	WAMANAGER_CICLO_PRELIEVO_PALL_RUN:
		IF Mission^.State = MISSION_STATE_NOP OR Mission^.State = MISSION_STATE_DEPOSITO_FALDA_END THEN
			QuotaFuoriIngombro_Z_AVUOTO_CCENTRALE := 0;
			QuotaFuoriIngombro_Z_ConPALLET := 0;
			(* Valuto gli ostacoli *)	
			FOR f:=1 TO MAXFOOTPRINT DO	
				IF QuotaFuoriIngombro_Z_AVUOTO_CCENTRALE <= WorkFootPrint^[f].Z + WorkFootPrint^[f].ZDim + TCPParameter.Z + OffsetSicurezza.Avuoto THEN
					QuotaFuoriIngombro_Z_AVUOTO_CCENTRALE := WorkFootPrint^[f].Z + WorkFootPrint^[f].ZDim + TCPParameter.Z + OffsetSicurezza.Avuoto;
				END_IF
				IF Mission^.TPick = TPICK_PALLET THEN
					IF QuotaFuoriIngombro_Z_ConPALLET <= WorkFootPrint^[f].Z + WorkFootPrint^[f].ZDim + Dimensione_Z_ElementoInPresaX_Ingombro + OffsetSicurezza.ConPallet THEN
						QuotaFuoriIngombro_Z_ConPALLET := WorkFootPrint^[f].Z + WorkFootPrint^[f].ZDim + Dimensione_Z_ElementoInPresaX_Ingombro + OffsetSicurezza.ConPallet;
					END_IF
				END_IF
			END_FOR
			(* Valuto le aree *)
			FOR a:=1 TO MAXAREA DO
				AltezzaDiIngombroArea_CCENTRALE := 0;
				IF WorkAreaState^[a].H > WorkAreaState^[a].HPL THEN
					AltezzaDiIngombroArea_CCENTRALE := WorkAreaState^[a].H;
				ELSE
					AltezzaDiIngombroArea_CCENTRALE := WorkAreaState^[a].HPL;
				END_IF
				(* Se ho la postazione falde e/o catasta vuoti con riscontri fissi metto la quota fissa di altezza della postazione all'altezza massima*)
				IF WorkArea^[a].Typology = TYPOLOGY_LAYER THEN
					AltezzaDiIngombroArea_CCENTRALE := ALTEZZA_CATASTA_FALDE;
				ELSIF  WorkArea^[a].Typology <> TYPOLOGY_STACK AND CATASTA_VUOTI_CON_RISCONTRI_FISSI THEN
					AltezzaDiIngombroArea_CCENTRALE := ALTEZZA_CATASTA_VUOTI;
				END_IF
				IF QuotaFuoriIngombro_Z_AVUOTO_CCENTRALE <= AltezzaDiIngombroArea_CCENTRALE + TCPParameter.Z + OffsetSicurezza.Avuoto THEN
					QuotaFuoriIngombro_Z_AVUOTO_CCENTRALE := AltezzaDiIngombroArea_CCENTRALE + TCPParameter.Z + OffsetSicurezza.Avuoto;
				END_IF
				IF QuotaFuoriIngombro_Z_ConPALLET <= AltezzaDiIngombroArea_CCENTRALE + Dimensione_Z_ElementoInPresaX_Ingombro + OffsetSicurezza.ConPallet THEN
					QuotaFuoriIngombro_Z_ConPALLET := AltezzaDiIngombroArea_CCENTRALE + Dimensione_Z_ElementoInPresaX_Ingombro + OffsetSicurezza.ConPallet;
				END_IF
			END_FOR
			(* Valuto I Pick-Point *)
			(*CASE TIPO_RIBALTINO OF
				RIBALTINO_DOPO_SQUADRO:
					FOR P:=1 TO MAXPICKPOINT DO
						AltezzaDiIngombroPuntiPrelievo := 0;
						IF  WorkPickPoint^[P].Zh + WorkPickPointState^[P].ZDim >= WorkPickPointDimension[P].Zdim THEN // Se Altezza orrizzontale Ribaltino + Zpacco >= Ingombro Verticale Ribaltino
							AltezzaDiIngombroPuntiPrelievo := WorkPickPoint^[P].Zh + WorkPickPointState^[P].ZDim;
						END_IF
						IF WorkPickPoint^[P].Zv + WorkPickPointState^[P].ZTilter + WorkPickPointState^[P].YDim >= WorkPickPointDimension[P].Zdim THEN // Se Altezza Vertivale Ribaltino + Quota Fermo + Ypacco >= Ingombro Verticale Ribaltino
							AltezzaDiIngombroPuntiPrelievo := WorkPickPoint^[P].Zv + WorkPickPointState^[P].ZTilter + WorkPickPointState^[P].YDim;
						END_IF
						IF WorkPickPointDimension[P].Zdim >= AltezzaDiIngombroPuntiPrelievo THEN //Se Ingombro Verticale Ribaltino >= Dell'ingombro valutato sopra
							AltezzaDiIngombroPuntiPrelievo := WorkPickPointDimension[P].Zdim;
						END_IF
						IF QuotaFuoriIngombro_Z_AVUOTO_CCENTRALE <= AltezzaDiIngombroPuntiPrelievo + TCPParameter.Z + OffsetSicurezza.Avuoto THEN //Se Quota fuori ingombro <= dell' ingombro del punto di prelievo
							QuotaFuoriIngombro_Z_AVUOTO_CCENTRALE := AltezzaDiIngombroPuntiPrelievo + TCPParameter.Z + OffsetSicurezza.Avuoto;
						END_IF				
					END_FOR
				RIBALTINO_DIRETTO :
					FOR P:=1 TO MAXPICKPOINT DO
						AltezzaDiIngombroPuntiPrelievo := 0;
						IF  WorkPickPoint^[P].Zh + WorkPickPointState^[P].ZDim >= WorkPickPointDimension[P].Zdim THEN // Se Altezza orrizzontale Ribaltino + Zpacco >= Ingombro Verticale Ribaltino
							AltezzaDiIngombroPuntiPrelievo := WorkPickPoint^[P].Zh + WorkPickPointState^[P].ZDim;
						END_IF
						IF WorkPickPoint^[P].Zv + WorkPickPointState^[P].ZTilter + WorkPickPointState^[P].XDim >= WorkPickPointDimension[P].Zdim THEN // Se Altezza Vertivale Ribaltino + Quota Fermo + Ypacco >= Ingombro Verticale Ribaltino
							AltezzaDiIngombroPuntiPrelievo := WorkPickPoint^[P].Zv + WorkPickPointState^[P].ZTilter + WorkPickPointState^[P].XDim;
						END_IF
						IF WorkPickPointDimension[P].Zdim >= AltezzaDiIngombroPuntiPrelievo THEN //Se Ingombro Verticale Ribaltino >= Dell'ingombro valutato sopra
							AltezzaDiIngombroPuntiPrelievo := WorkPickPointDimension[P].Zdim;
						END_IF
						IF QuotaFuoriIngombro_Z_AVUOTO_CCENTRALE <= AltezzaDiIngombroPuntiPrelievo + TCPParameter.Z + OffsetSicurezza.Avuoto THEN //Se Quota fuori ingombro <= dell' ingombro del punto di prelievo
							QuotaFuoriIngombro_Z_AVUOTO_CCENTRALE := AltezzaDiIngombroPuntiPrelievo + TCPParameter.Z + OffsetSicurezza.Avuoto;
						END_IF				
					END_FOR
			END_CASE*)
			
			(*IF Mission^.TPick = TPICK_PALLET THEN
				Traiettoria^.PassModePoint_Z_Enable[1] := TRUE; // traslazione verso l'alto e verticale.....inizio degli altri movimenti 200 mm prima dela fine
				Traiettoria^.PassModePoint_Z[1] := QuotaFuoriIngombro_Z_AVUOTO_CCENTRALE - OffsetPassMode.Z;
				Traiettoria^.PassModePoint_X_Enable[1] := TRUE;	
				IF ModuleAX_X^.Ax^.Status.ActPosition >= Mission^.XPick THEN			// se la posizione attuale in X è MAGGIORE della posizione di destinazione
					Traiettoria^.PassModePoint_X[1] := Mission^.XPick + OffsetPassMode.X;			
				ELSE																	// se la posizione attuale in X è MINORE della posizione di destinazione
					Traiettoria^.PassModePoint_X[1] := Mission^.XPick - OffsetPassMode.X;			
				END_IF			
				Traiettoria^.PassModePoint_Y_Enable[1] := TRUE;
				Traiettoria^.PassModePoint_Y[1] := 0;			// inizio degli altri movimenti in corrispondenza della posizione attuale
				Traiettoria^.PassModePoint_J_Enable[1] := TRUE;
				Traiettoria^.PassModePoint_J[1] := 0;			// inizio degli altri movimenti in corrispondenza della posizione attuale
				Traiettoria^.PassModePoint_K_Enable[1] := TRUE;
				Traiettoria^.PassModePoint_K[1] := 0;			// inizio degli altri movimenti in corrispondenza della posizione attuale
			END_IF*)
		END_IF //riferito all'IF dello stato della missione	
														
	WAMANAGER_CICLO_PRELIEVO_PALL_END,						
		
	WAMANAGER_CICLO_DEPOSITO_PALL_RUN:
		IF Mission^.State = MISSION_STATE_NOP OR Mission^.State = MISSION_STATE_PRELIEVO_PALLET_END THEN
			QuotaFuoriIngombro_Z_AVUOTO_CCENTRALE := 0;
			QuotaFuoriIngombro_Z_ConPALLET := 0;
			(* Valuto gli ostacoli x la quota fuori ingombro*)	
			FOR f:=1 TO MAXFOOTPRINT DO	
				IF QuotaFuoriIngombro_Z_AVUOTO_CCENTRALE <= WorkFootPrint^[f].Z + WorkFootPrint^[f].ZDim + TCPParameter.Z + OffsetSicurezza.Avuoto THEN
					QuotaFuoriIngombro_Z_AVUOTO_CCENTRALE := WorkFootPrint^[f].Z + WorkFootPrint^[f].ZDim + TCPParameter.Z + OffsetSicurezza.Avuoto;
				END_IF
				IF QuotaFuoriIngombro_Z_ConPALLET <= WorkFootPrint^[f].Z + WorkFootPrint^[f].ZDim + Dimensione_Z_ElementoInPresaX_Ingombro + OffsetSicurezza.ConPallet THEN
					QuotaFuoriIngombro_Z_ConPALLET := WorkFootPrint^[f].Z + WorkFootPrint^[f].ZDim + Dimensione_Z_ElementoInPresaX_Ingombro + OffsetSicurezza.ConPallet;
				END_IF
			END_FOR
			(* Valuto le aree x la quota fuori ingombro *)
			FOR a:=1 TO MAXAREA DO
				AltezzaDiIngombroArea_CCENTRALE := 0;
				IF WorkAreaState^[a].H > WorkAreaState^[a].HPL THEN
					AltezzaDiIngombroArea_CCENTRALE := WorkAreaState^[a].H;
				ELSE
					AltezzaDiIngombroArea_CCENTRALE := WorkAreaState^[a].HPL;
				END_IF
				(* Se ho la postazione falde e/o catasta vuoti con riscontri fissi metto la quota fissa di altezza della postazione all'altezza massima*)
				IF WorkArea^[a].Typology = TYPOLOGY_LAYER THEN
					AltezzaDiIngombroArea_CCENTRALE := ALTEZZA_CATASTA_FALDE;
				ELSIF  WorkArea^[a].Typology <> TYPOLOGY_STACK AND CATASTA_VUOTI_CON_RISCONTRI_FISSI THEN
					AltezzaDiIngombroArea_CCENTRALE := ALTEZZA_CATASTA_VUOTI;
				END_IF
				IF QuotaFuoriIngombro_Z_AVUOTO_CCENTRALE <= AltezzaDiIngombroArea_CCENTRALE + TCPParameter.Z + OffsetSicurezza.Avuoto THEN
					QuotaFuoriIngombro_Z_AVUOTO_CCENTRALE := AltezzaDiIngombroArea_CCENTRALE + TCPParameter.Z + OffsetSicurezza.Avuoto;
				END_IF
				IF QuotaFuoriIngombro_Z_ConPALLET <= AltezzaDiIngombroArea_CCENTRALE + Dimensione_Z_ElementoInPresaX_Ingombro + OffsetSicurezza.ConPallet THEN
					QuotaFuoriIngombro_Z_ConPALLET := AltezzaDiIngombroArea_CCENTRALE + Dimensione_Z_ElementoInPresaX_Ingombro + OffsetSicurezza.ConPallet;
				END_IF
			END_FOR
			(* Valuto I Pick-Point *)
			(* Valuto I Pick-Point *)
			(*CASE TIPO_RIBALTINO OF
				RIBALTINO_DOPO_SQUADRO:
					FOR P:=1 TO MAXPICKPOINT DO
						AltezzaDiIngombroPuntiPrelievo := 0;
						IF  WorkPickPoint^[P].Zh + WorkPickPointState^[P].ZDim >= WorkPickPointDimension[P].Zdim THEN // Se Altezza orrizzontale Ribaltino + Zpacco >= Ingombro Verticale Ribaltino
							AltezzaDiIngombroPuntiPrelievo := WorkPickPoint^[P].Zh + WorkPickPointState^[P].ZDim;
						END_IF
						IF WorkPickPoint^[P].Zv + WorkPickPointState^[P].ZTilter + WorkPickPointState^[P].YDim >= WorkPickPointDimension[P].Zdim THEN // Se Altezza Vertivale Ribaltino + Quota Fermo + Ypacco >= Ingombro Verticale Ribaltino
							AltezzaDiIngombroPuntiPrelievo := WorkPickPoint^[P].Zv + WorkPickPointState^[P].ZTilter + WorkPickPointState^[P].YDim;
						END_IF
						IF WorkPickPointDimension[P].Zdim >= AltezzaDiIngombroPuntiPrelievo THEN //Se Ingombro Verticale Ribaltino >= Dell'ingombro valutato sopra
							AltezzaDiIngombroPuntiPrelievo := WorkPickPointDimension[P].Zdim;
						END_IF
						IF QuotaFuoriIngombro_Z_AVUOTO_CCENTRALE <= AltezzaDiIngombroPuntiPrelievo + TCPParameter.Z + OffsetSicurezza.Avuoto THEN //Se Quota fuori ingombro <= dell' ingombro del punto di prelievo
							QuotaFuoriIngombro_Z_AVUOTO_CCENTRALE := AltezzaDiIngombroPuntiPrelievo + TCPParameter.Z + OffsetSicurezza.Avuoto;
						END_IF
						IF QuotaFuoriIngombro_Z_ConPALLET <= AltezzaDiIngombroPuntiPrelievo + TCPParameter.Z + OffsetSicurezza.ConPallet THEN //Se Quota fuori ingombro <= dell' ingombro del punto di prelievo
							QuotaFuoriIngombro_Z_ConPALLET := AltezzaDiIngombroPuntiPrelievo + TCPParameter.Z + OffsetSicurezza.ConPallet;
						END_IF
					END_FOR
				RIBALTINO_DIRETTO :
					FOR P:=1 TO MAXPICKPOINT DO
						AltezzaDiIngombroPuntiPrelievo := 0;
						IF  WorkPickPoint^[P].Zh + WorkPickPointState^[P].ZDim >= WorkPickPointDimension[P].Zdim THEN // Se Altezza orrizzontale Ribaltino + Zpacco >= Ingombro Verticale Ribaltino
							AltezzaDiIngombroPuntiPrelievo := WorkPickPoint^[P].Zh + WorkPickPointState^[P].ZDim;
						END_IF
						IF WorkPickPoint^[P].Zv + WorkPickPointState^[P].ZTilter + WorkPickPointState^[P].XDim >= WorkPickPointDimension[P].Zdim THEN // Se Altezza Vertivale Ribaltino + Quota Fermo + Ypacco >= Ingombro Verticale Ribaltino
							AltezzaDiIngombroPuntiPrelievo := WorkPickPoint^[P].Zv + WorkPickPointState^[P].ZTilter + WorkPickPointState^[P].XDim;
						END_IF
						IF WorkPickPointDimension[P].Zdim >= AltezzaDiIngombroPuntiPrelievo THEN //Se Ingombro Verticale Ribaltino >= Dell'ingombro valutato sopra
							AltezzaDiIngombroPuntiPrelievo := WorkPickPointDimension[P].Zdim;
						END_IF
						IF QuotaFuoriIngombro_Z_AVUOTO_CCENTRALE <= AltezzaDiIngombroPuntiPrelievo + TCPParameter.Z + OffsetSicurezza.Avuoto THEN //Se Quota fuori ingombro <= dell' ingombro del punto di prelievo
							QuotaFuoriIngombro_Z_AVUOTO_CCENTRALE := AltezzaDiIngombroPuntiPrelievo + TCPParameter.Z + OffsetSicurezza.Avuoto;
						END_IF	
						IF QuotaFuoriIngombro_Z_ConPALLET <= AltezzaDiIngombroPuntiPrelievo + TCPParameter.Z + OffsetSicurezza.ConPallet THEN //Se Quota fuori ingombro <= dell' ingombro del punto di prelievo
							QuotaFuoriIngombro_Z_ConPALLET := AltezzaDiIngombroPuntiPrelievo + TCPParameter.Z + OffsetSicurezza.ConPallet;
						END_IF			
					END_FOR
			END_CASE*)
					
		END_IF //riferito all'IF dello stato della missione	
		
			
	WAMANAGER_CICLO_DEPOSITO_PALL_END,
	
	WAMANAGER_CICLO_FALDA_VUOTI_INIT,
	
	WAMANAGER_CICLO_PRELIEVO_FALDA_VUOTI_RUN:
		IF Mission^.State = MISSION_STATE_NOP THEN
			QuotaFuoriIngombro_Z_AVUOTO_CCENTRALE := 0;
			QuotaFuoriIngombro_Z_ConFALDA := 0;
			(* Valuto gli ostacoli *)	
			FOR f:=1 TO MAXFOOTPRINT DO	
				IF QuotaFuoriIngombro_Z_AVUOTO_CCENTRALE <= WorkFootPrint^[f].Z + WorkFootPrint^[f].ZDim + TCPParameter.Z + OffsetSicurezza.Avuoto THEN
					QuotaFuoriIngombro_Z_AVUOTO_CCENTRALE := WorkFootPrint^[f].Z + WorkFootPrint^[f].ZDim + TCPParameter.Z + OffsetSicurezza.Avuoto;
				END_IF
			END_FOR
			(* Valuto le aree *)
			FOR a:=1 TO MAXAREA DO
				AltezzaDiIngombroArea_CCENTRALE := 0;
				IF WorkAreaState^[a].H > WorkAreaState^[a].HPL THEN
					AltezzaDiIngombroArea_CCENTRALE := WorkAreaState^[a].H;
				ELSE
					AltezzaDiIngombroArea_CCENTRALE := WorkAreaState^[a].HPL;
				END_IF
				(* Se ho la postazione falde e/o catasta vuoti con riscontri fissi metto la quota fissa di altezza della postazione all'altezza massima*)
				IF WorkArea^[a].Typology = TYPOLOGY_LAYER THEN
					AltezzaDiIngombroArea_CCENTRALE := ALTEZZA_CATASTA_FALDE;
				ELSIF  WorkArea^[a].Typology <> TYPOLOGY_STACK AND CATASTA_VUOTI_CON_RISCONTRI_FISSI THEN
					AltezzaDiIngombroArea_CCENTRALE := ALTEZZA_CATASTA_VUOTI;
				END_IF
				IF QuotaFuoriIngombro_Z_AVUOTO_CCENTRALE <= AltezzaDiIngombroArea_CCENTRALE + TCPParameter.Z + OffsetSicurezza.Avuoto THEN
					QuotaFuoriIngombro_Z_AVUOTO_CCENTRALE := AltezzaDiIngombroArea_CCENTRALE + TCPParameter.Z + OffsetSicurezza.Avuoto;
				END_IF
			END_FOR
			(* Valuto I Pick-Point *)
			(*CASE TIPO_RIBALTINO OF
				RIBALTINO_DOPO_SQUADRO:
					FOR P:=1 TO MAXPICKPOINT DO
						AltezzaDiIngombroPuntiPrelievo := 0;
						IF  WorkPickPoint^[P].Zh + WorkPickPointState^[P].ZDim >= WorkPickPointDimension[P].Zdim THEN // Se Altezza orrizzontale Ribaltino + Zpacco >= Ingombro Verticale Ribaltino
							AltezzaDiIngombroPuntiPrelievo := WorkPickPoint^[P].Zh + WorkPickPointState^[P].ZDim;
						END_IF
						IF WorkPickPoint^[P].Zv + WorkPickPointState^[P].ZTilter + WorkPickPointState^[P].YDim >= WorkPickPointDimension[P].Zdim THEN // Se Altezza Vertivale Ribaltino + Quota Fermo + Ypacco >= Ingombro Verticale Ribaltino
							AltezzaDiIngombroPuntiPrelievo := WorkPickPoint^[P].Zv + WorkPickPointState^[P].ZTilter + WorkPickPointState^[P].YDim;
						END_IF
						IF WorkPickPointDimension[P].Zdim >= AltezzaDiIngombroPuntiPrelievo THEN //Se Ingombro Verticale Ribaltino >= Dell'ingombro valutato sopra
							AltezzaDiIngombroPuntiPrelievo := WorkPickPointDimension[P].Zdim;
						END_IF
						IF QuotaFuoriIngombro_Z_AVUOTO_CCENTRALE <= AltezzaDiIngombroPuntiPrelievo + TCPParameter.Z + OffsetSicurezza.Avuoto THEN //Se Quota fuori ingombro <= dell' ingombro del punto di prelievo
							QuotaFuoriIngombro_Z_AVUOTO_CCENTRALE := AltezzaDiIngombroPuntiPrelievo + TCPParameter.Z + OffsetSicurezza.Avuoto;
						END_IF				
					END_FOR
				RIBALTINO_DIRETTO :
					FOR P:=1 TO MAXPICKPOINT DO
						AltezzaDiIngombroPuntiPrelievo := 0;
						IF  WorkPickPoint^[P].Zh + WorkPickPointState^[P].ZDim >= WorkPickPointDimension[P].Zdim THEN // Se Altezza orrizzontale Ribaltino + Zpacco >= Ingombro Verticale Ribaltino
							AltezzaDiIngombroPuntiPrelievo := WorkPickPoint^[P].Zh + WorkPickPointState^[P].ZDim;
						END_IF
						IF WorkPickPoint^[P].Zv + WorkPickPointState^[P].ZTilter + WorkPickPointState^[P].XDim >= WorkPickPointDimension[P].Zdim THEN // Se Altezza Vertivale Ribaltino + Quota Fermo + Ypacco >= Ingombro Verticale Ribaltino
							AltezzaDiIngombroPuntiPrelievo := WorkPickPoint^[P].Zv + WorkPickPointState^[P].ZTilter + WorkPickPointState^[P].XDim;
						END_IF
						IF WorkPickPointDimension[P].Zdim >= AltezzaDiIngombroPuntiPrelievo THEN //Se Ingombro Verticale Ribaltino >= Dell'ingombro valutato sopra
							AltezzaDiIngombroPuntiPrelievo := WorkPickPointDimension[P].Zdim;
						END_IF
						IF QuotaFuoriIngombro_Z_AVUOTO_CCENTRALE <= AltezzaDiIngombroPuntiPrelievo + TCPParameter.Z + OffsetSicurezza.Avuoto THEN //Se Quota fuori ingombro <= dell' ingombro del punto di prelievo
							QuotaFuoriIngombro_Z_AVUOTO_CCENTRALE := AltezzaDiIngombroPuntiPrelievo + TCPParameter.Z + OffsetSicurezza.Avuoto;
						END_IF				
					END_FOR
			END_CASE*)
			QuotaFuoriIngombro_Z_ConFALDA := QuotaFuoriIngombro_Z_AVUOTO_CCENTRALE;
			
		END_IF //riferito all'IF dello stato della missione	
					
	WAMANAGER_CICLO_PRELIEVO_FALDA_VUOTI_END,
		
	WAMANAGER_CICLO_DEPOSITO_FALDA_VUOTI_RUN:
		IF Mission^.State = MISSION_STATE_NOP OR Mission^.State = MISSION_STATE_PRELIEVO_FALDA_END THEN
			QuotaFuoriIngombro_Z_AVUOTO_CCENTRALE := 0;
			QuotaFuoriIngombro_Z_ConFALDA := 0;
			(* Valuto gli ostacoli *)	
			FOR f:=1 TO MAXFOOTPRINT DO	
				IF QuotaFuoriIngombro_Z_AVUOTO_CCENTRALE <= WorkFootPrint^[f].Z + WorkFootPrint^[f].ZDim + TCPParameter.Z + OffsetSicurezza.Avuoto THEN
					QuotaFuoriIngombro_Z_AVUOTO_CCENTRALE := WorkFootPrint^[f].Z + WorkFootPrint^[f].ZDim + TCPParameter.Z + OffsetSicurezza.Avuoto;
				END_IF
			END_FOR
			(* Valuto le aree *)
			FOR a:=1 TO MAXAREA DO
				AltezzaDiIngombroArea_CCENTRALE := 0;
				IF WorkAreaState^[a].H > WorkAreaState^[a].HPL THEN
					AltezzaDiIngombroArea_CCENTRALE := WorkAreaState^[a].H;
				ELSE
					AltezzaDiIngombroArea_CCENTRALE := WorkAreaState^[a].HPL;
				END_IF
				(* Se ho la postazione falde e/o catasta vuoti con riscontri fissi metto la quota fissa di altezza della postazione all'altezza massima*)
				IF WorkArea^[a].Typology = TYPOLOGY_LAYER THEN
					AltezzaDiIngombroArea_CCENTRALE := ALTEZZA_CATASTA_FALDE;
				ELSIF  WorkArea^[a].Typology <> TYPOLOGY_STACK AND CATASTA_VUOTI_CON_RISCONTRI_FISSI THEN
					AltezzaDiIngombroArea_CCENTRALE := ALTEZZA_CATASTA_VUOTI;
				END_IF
				IF QuotaFuoriIngombro_Z_AVUOTO_CCENTRALE <= AltezzaDiIngombroArea_CCENTRALE + TCPParameter.Z + OffsetSicurezza.Avuoto THEN
					QuotaFuoriIngombro_Z_AVUOTO_CCENTRALE := AltezzaDiIngombroArea_CCENTRALE + TCPParameter.Z + OffsetSicurezza.Avuoto;
				END_IF
			END_FOR
			(* Valuto I Pick-Point *)
			(*CASE TIPO_RIBALTINO OF
				RIBALTINO_DOPO_SQUADRO:
					FOR P:=1 TO MAXPICKPOINT DO
						AltezzaDiIngombroPuntiPrelievo := 0;
						IF  WorkPickPoint^[P].Zh + WorkPickPointState^[P].ZDim >= WorkPickPointDimension[P].Zdim THEN // Se Altezza orrizzontale Ribaltino + Zpacco >= Ingombro Verticale Ribaltino
							AltezzaDiIngombroPuntiPrelievo := WorkPickPoint^[P].Zh + WorkPickPointState^[P].ZDim;
						END_IF
						IF WorkPickPoint^[P].Zv + WorkPickPointState^[P].ZTilter + WorkPickPointState^[P].YDim >= WorkPickPointDimension[P].Zdim THEN // Se Altezza Vertivale Ribaltino + Quota Fermo + Ypacco >= Ingombro Verticale Ribaltino
							AltezzaDiIngombroPuntiPrelievo := WorkPickPoint^[P].Zv + WorkPickPointState^[P].ZTilter + WorkPickPointState^[P].YDim;
						END_IF
						IF WorkPickPointDimension[P].Zdim >= AltezzaDiIngombroPuntiPrelievo THEN //Se Ingombro Verticale Ribaltino >= Dell'ingombro valutato sopra
							AltezzaDiIngombroPuntiPrelievo := WorkPickPointDimension[P].Zdim;
						END_IF
						IF QuotaFuoriIngombro_Z_AVUOTO_CCENTRALE <= AltezzaDiIngombroPuntiPrelievo + TCPParameter.Z + OffsetSicurezza.Avuoto THEN //Se Quota fuori ingombro <= dell' ingombro del punto di prelievo
							QuotaFuoriIngombro_Z_AVUOTO_CCENTRALE := AltezzaDiIngombroPuntiPrelievo + TCPParameter.Z + OffsetSicurezza.Avuoto;
						END_IF				
					END_FOR
				RIBALTINO_DIRETTO :
					FOR P:=1 TO MAXPICKPOINT DO
						AltezzaDiIngombroPuntiPrelievo := 0;
						IF  WorkPickPoint^[P].Zh + WorkPickPointState^[P].ZDim >= WorkPickPointDimension[P].Zdim THEN // Se Altezza orrizzontale Ribaltino + Zpacco >= Ingombro Verticale Ribaltino
							AltezzaDiIngombroPuntiPrelievo := WorkPickPoint^[P].Zh + WorkPickPointState^[P].ZDim;
						END_IF
						IF WorkPickPoint^[P].Zv + WorkPickPointState^[P].ZTilter + WorkPickPointState^[P].XDim >= WorkPickPointDimension[P].Zdim THEN // Se Altezza Vertivale Ribaltino + Quota Fermo + Ypacco >= Ingombro Verticale Ribaltino
							AltezzaDiIngombroPuntiPrelievo := WorkPickPoint^[P].Zv + WorkPickPointState^[P].ZTilter + WorkPickPointState^[P].XDim;
						END_IF
						IF WorkPickPointDimension[P].Zdim >= AltezzaDiIngombroPuntiPrelievo THEN //Se Ingombro Verticale Ribaltino >= Dell'ingombro valutato sopra
							AltezzaDiIngombroPuntiPrelievo := WorkPickPointDimension[P].Zdim;
						END_IF
						IF QuotaFuoriIngombro_Z_AVUOTO_CCENTRALE <= AltezzaDiIngombroPuntiPrelievo + TCPParameter.Z + OffsetSicurezza.Avuoto THEN //Se Quota fuori ingombro <= dell' ingombro del punto di prelievo
							QuotaFuoriIngombro_Z_AVUOTO_CCENTRALE := AltezzaDiIngombroPuntiPrelievo + TCPParameter.Z + OffsetSicurezza.Avuoto;
						END_IF				
					END_FOR
			END_CASE*)
			QuotaFuoriIngombro_Z_ConFALDA := QuotaFuoriIngombro_Z_AVUOTO_CCENTRALE;
			
		END_IF //riferito all'IF dello stato della missione	
									
	WAMANAGER_CICLO_DEPOSITO_FALDA_VUOTI_END,*)
	
	WAMANAGER_CICLO_FALDA_INIT,
	
	WAMANAGER_CICLO_PRELIEVO_FALDA_RUN:
		IF Mission^.State = MISSION_STATE_NOP THEN
			QuotaFuoriIngombro_Z_AVUOTO_CCENTRALE := 0;
			QuotaFuoriIngombro_Z_ConFALDA := 0;
			(* Valuto gli ostacoli *)	
			FOR f:=1 TO MAXFOOTPRINT DO	
				IF QuotaFuoriIngombro_Z_AVUOTO_CCENTRALE <= WorkFootPrint^[f].Z + WorkFootPrint^[f].ZDim + TCPParameter.Z + OffsetSicurezza.Avuoto THEN
					QuotaFuoriIngombro_Z_AVUOTO_CCENTRALE := WorkFootPrint^[f].Z + WorkFootPrint^[f].ZDim + TCPParameter.Z + OffsetSicurezza.Avuoto;
				END_IF
			END_FOR
			(* Valuto le aree *)
			FOR a:=1 TO MAXAREA DO
				AltezzaDiIngombroArea_CCENTRALE := 0;
				IF WorkAreaState^[a].H > WorkAreaState^[a].HPL THEN
					AltezzaDiIngombroArea_CCENTRALE := WorkAreaState^[a].H;
				ELSE
					AltezzaDiIngombroArea_CCENTRALE := WorkAreaState^[a].HPL;
				END_IF
				IF QuotaFuoriIngombro_Z_AVUOTO_CCENTRALE <= AltezzaDiIngombroArea_CCENTRALE + TCPParameter.Z + OffsetSicurezza.Avuoto THEN
					QuotaFuoriIngombro_Z_AVUOTO_CCENTRALE := AltezzaDiIngombroArea_CCENTRALE + TCPParameter.Z + OffsetSicurezza.Avuoto;
				END_IF
			END_FOR
			(* Valuto I Pick-Point *)
			(*CASE TIPO_RIBALTINO OF
				RIBALTINO_DOPO_SQUADRO:
					FOR P:=1 TO MAXPICKPOINT DO
						AltezzaDiIngombroPuntiPrelievo := 0;
						IF  WorkPickPoint^[P].Zh + WorkPickPointState^[P].ZDim >= WorkPickPointDimension[P].Zdim THEN // Se Altezza orrizzontale Ribaltino + Zpacco >= Ingombro Verticale Ribaltino
							AltezzaDiIngombroPuntiPrelievo := WorkPickPoint^[P].Zh + WorkPickPointState^[P].ZDim;
						END_IF
						IF WorkPickPoint^[P].Zv + WorkPickPointState^[P].ZTilter + WorkPickPointState^[P].YDim >= WorkPickPointDimension[P].Zdim THEN // Se Altezza Vertivale Ribaltino + Quota Fermo + Ypacco >= Ingombro Verticale Ribaltino
							AltezzaDiIngombroPuntiPrelievo := WorkPickPoint^[P].Zv + WorkPickPointState^[P].ZTilter + WorkPickPointState^[P].YDim;
						END_IF
						IF WorkPickPointDimension[P].Zdim >= AltezzaDiIngombroPuntiPrelievo THEN //Se Ingombro Verticale Ribaltino >= Dell'ingombro valutato sopra
							AltezzaDiIngombroPuntiPrelievo := WorkPickPointDimension[P].Zdim;
						END_IF
						IF QuotaFuoriIngombro_Z_AVUOTO_CCENTRALE <= AltezzaDiIngombroPuntiPrelievo + TCPParameter.Z + OffsetSicurezza.Avuoto THEN //Se Quota fuori ingombro <= dell' ingombro del punto di prelievo
							QuotaFuoriIngombro_Z_AVUOTO_CCENTRALE := AltezzaDiIngombroPuntiPrelievo + TCPParameter.Z + OffsetSicurezza.Avuoto;
						END_IF				
					END_FOR
				RIBALTINO_DIRETTO :
					FOR P:=1 TO MAXPICKPOINT DO
						AltezzaDiIngombroPuntiPrelievo := 0;
						IF  WorkPickPoint^[P].Zh + WorkPickPointState^[P].ZDim >= WorkPickPointDimension[P].Zdim THEN // Se Altezza orrizzontale Ribaltino + Zpacco >= Ingombro Verticale Ribaltino
							AltezzaDiIngombroPuntiPrelievo := WorkPickPoint^[P].Zh + WorkPickPointState^[P].ZDim;
						END_IF
						IF WorkPickPoint^[P].Zv + WorkPickPointState^[P].ZTilter + WorkPickPointState^[P].XDim >= WorkPickPointDimension[P].Zdim THEN // Se Altezza Vertivale Ribaltino + Quota Fermo + Ypacco >= Ingombro Verticale Ribaltino
							AltezzaDiIngombroPuntiPrelievo := WorkPickPoint^[P].Zv + WorkPickPointState^[P].ZTilter + WorkPickPointState^[P].XDim;
						END_IF
						IF WorkPickPointDimension[P].Zdim >= AltezzaDiIngombroPuntiPrelievo THEN //Se Ingombro Verticale Ribaltino >= Dell'ingombro valutato sopra
							AltezzaDiIngombroPuntiPrelievo := WorkPickPointDimension[P].Zdim;
						END_IF
						IF QuotaFuoriIngombro_Z_AVUOTO_CCENTRALE <= AltezzaDiIngombroPuntiPrelievo + TCPParameter.Z + OffsetSicurezza.Avuoto THEN //Se Quota fuori ingombro <= dell' ingombro del punto di prelievo
							QuotaFuoriIngombro_Z_AVUOTO_CCENTRALE := AltezzaDiIngombroPuntiPrelievo + TCPParameter.Z + OffsetSicurezza.Avuoto;
						END_IF				
					END_FOR
			END_CASE*)
			QuotaFuoriIngombro_Z_ConFALDA := QuotaFuoriIngombro_Z_AVUOTO_CCENTRALE;
			
		END_IF //riferito all'IF dello stato della missione	
																
	WAMANAGER_CICLO_PRELIEVO_FALDA_END,
			
	WAMANAGER_CICLO_DEPOSITO_FALDA_RUN:
		IF Mission^.State = MISSION_STATE_NOP OR Mission^.State = MISSION_STATE_PRELIEVO_FALDA_END THEN
			QuotaFuoriIngombro_Z_AVUOTO_CCENTRALE := 0;
			QuotaFuoriIngombro_Z_ConFALDA := 0;
			(* Valuto gli ostacoli *)	
			FOR f:=1 TO MAXFOOTPRINT DO	
				IF QuotaFuoriIngombro_Z_AVUOTO_CCENTRALE <= WorkFootPrint^[f].Z + WorkFootPrint^[f].ZDim + TCPParameter.Z + OffsetSicurezza.Avuoto THEN
					QuotaFuoriIngombro_Z_AVUOTO_CCENTRALE := WorkFootPrint^[f].Z + WorkFootPrint^[f].ZDim + TCPParameter.Z + OffsetSicurezza.Avuoto;
				END_IF
			END_FOR
			(* Valuto le aree *)
			FOR a:=1 TO MAXAREA DO
				AltezzaDiIngombroArea_CCENTRALE := 0;
				IF WorkAreaState^[a].H > WorkAreaState^[a].HPL THEN
					AltezzaDiIngombroArea_CCENTRALE := WorkAreaState^[a].H;
				ELSE
					AltezzaDiIngombroArea_CCENTRALE := WorkAreaState^[a].HPL;
				END_IF
				IF QuotaFuoriIngombro_Z_AVUOTO_CCENTRALE <= AltezzaDiIngombroArea_CCENTRALE + TCPParameter.Z + OffsetSicurezza.Avuoto THEN
					QuotaFuoriIngombro_Z_AVUOTO_CCENTRALE := AltezzaDiIngombroArea_CCENTRALE + TCPParameter.Z + OffsetSicurezza.Avuoto;
				END_IF
			END_FOR
			(* Valuto I Pick-Point *)
			(*CASE TIPO_RIBALTINO OF
				RIBALTINO_DOPO_SQUADRO:
					FOR P:=1 TO MAXPICKPOINT DO
						AltezzaDiIngombroPuntiPrelievo := 0;
						IF  WorkPickPoint^[P].Zh + WorkPickPointState^[P].ZDim >= WorkPickPointDimension[P].Zdim THEN // Se Altezza orrizzontale Ribaltino + Zpacco >= Ingombro Verticale Ribaltino
							AltezzaDiIngombroPuntiPrelievo := WorkPickPoint^[P].Zh + WorkPickPointState^[P].ZDim;
						END_IF
						IF WorkPickPoint^[P].Zv + WorkPickPointState^[P].ZTilter + WorkPickPointState^[P].YDim >= WorkPickPointDimension[P].Zdim THEN // Se Altezza Vertivale Ribaltino + Quota Fermo + Ypacco >= Ingombro Verticale Ribaltino
							AltezzaDiIngombroPuntiPrelievo := WorkPickPoint^[P].Zv + WorkPickPointState^[P].ZTilter + WorkPickPointState^[P].YDim;
						END_IF
						IF WorkPickPointDimension[P].Zdim >= AltezzaDiIngombroPuntiPrelievo THEN //Se Ingombro Verticale Ribaltino >= Dell'ingombro valutato sopra
							AltezzaDiIngombroPuntiPrelievo := WorkPickPointDimension[P].Zdim;
						END_IF
						IF QuotaFuoriIngombro_Z_AVUOTO_CCENTRALE <= AltezzaDiIngombroPuntiPrelievo + TCPParameter.Z + OffsetSicurezza.Avuoto THEN //Se Quota fuori ingombro <= dell' ingombro del punto di prelievo
							QuotaFuoriIngombro_Z_AVUOTO_CCENTRALE := AltezzaDiIngombroPuntiPrelievo + TCPParameter.Z + OffsetSicurezza.Avuoto;
						END_IF				
					END_FOR
				RIBALTINO_DIRETTO :
					FOR P:=1 TO MAXPICKPOINT DO
						AltezzaDiIngombroPuntiPrelievo := 0;
						IF  WorkPickPoint^[P].Zh + WorkPickPointState^[P].ZDim >= WorkPickPointDimension[P].Zdim THEN // Se Altezza orrizzontale Ribaltino + Zpacco >= Ingombro Verticale Ribaltino
							AltezzaDiIngombroPuntiPrelievo := WorkPickPoint^[P].Zh + WorkPickPointState^[P].ZDim;
						END_IF
						IF WorkPickPoint^[P].Zv + WorkPickPointState^[P].ZTilter + WorkPickPointState^[P].XDim >= WorkPickPointDimension[P].Zdim THEN // Se Altezza Vertivale Ribaltino + Quota Fermo + Ypacco >= Ingombro Verticale Ribaltino
							AltezzaDiIngombroPuntiPrelievo := WorkPickPoint^[P].Zv + WorkPickPointState^[P].ZTilter + WorkPickPointState^[P].XDim;
						END_IF
						IF WorkPickPointDimension[P].Zdim >= AltezzaDiIngombroPuntiPrelievo THEN //Se Ingombro Verticale Ribaltino >= Dell'ingombro valutato sopra
							AltezzaDiIngombroPuntiPrelievo := WorkPickPointDimension[P].Zdim;
						END_IF
						IF QuotaFuoriIngombro_Z_AVUOTO_CCENTRALE <= AltezzaDiIngombroPuntiPrelievo + TCPParameter.Z + OffsetSicurezza.Avuoto THEN //Se Quota fuori ingombro <= dell' ingombro del punto di prelievo
							QuotaFuoriIngombro_Z_AVUOTO_CCENTRALE := AltezzaDiIngombroPuntiPrelievo + TCPParameter.Z + OffsetSicurezza.Avuoto;
						END_IF				
					END_FOR
			END_CASE*)
			QuotaFuoriIngombro_Z_ConFALDA := QuotaFuoriIngombro_Z_AVUOTO_CCENTRALE;
			
		END_IF //riferito all'IF dello stato della missione	
			
	//WAMANAGER_CICLO_DEPOSITO_FALDA_END,

	(*WAMANAGER_CICLO_PACCO_INIT,
	
	WAMANAGER_CICLO_PRELIEVO_PACCO_RUN:
		IF Mission^.State = MISSION_STATE_NOP THEN
			QuotaFuoriIngombro_Z_AVUOTO_CCENTRALE := 0;
			QuotaFuoriIngombro_Z_ConPEZZO := 0;
			(* Valuto gli ostacoli per calcolare il fuori ingombro di Z *)
			FOR f:=1 TO MAXFOOTPRINT DO	
				IF QuotaFuoriIngombro_Z_AVUOTO_CCENTRALE <= WorkFootPrint^[f].Z + WorkFootPrint^[f].ZDim + TCPParameter.Z + OffsetSicurezza.Avuoto THEN
					QuotaFuoriIngombro_Z_AVUOTO_CCENTRALE := WorkFootPrint^[f].Z + WorkFootPrint^[f].ZDim + TCPParameter.Z + OffsetSicurezza.Avuoto;
				END_IF
				IF QuotaFuoriIngombro_Z_ConPEZZO <= WorkFootPrint^[f].Z + WorkFootPrint^[f].ZDim + Dimensione_Z_ElementoInPresaX_Ingombro + OffsetSicurezza.ConPacco THEN
					QuotaFuoriIngombro_Z_ConPEZZO := WorkFootPrint^[f].Z + WorkFootPrint^[f].ZDim + Dimensione_Z_ElementoInPresaX_Ingombro + OffsetSicurezza.ConPacco;
				END_IF
			END_FOR
			(* Valuto le aree *)
			FOR a:=1 TO MAXAREA DO
				AltezzaDiIngombroArea_CCENTRALE := 0;
				IF WorkArea^[a].Typology <> TYPOLOGY_LAYER AND  WorkArea^[a].Typology <> TYPOLOGY_STACK THEN
					IF WorkAreaState^[a].H > WorkAreaState^[a].HPL THEN
						AltezzaDiIngombroArea_CCENTRALE := WorkAreaState^[a].H;
					ELSE
						AltezzaDiIngombroArea_CCENTRALE := WorkAreaState^[a].HPL;
					END_IF
					IF QuotaFuoriIngombro_Z_AVUOTO_CCENTRALE <= AltezzaDiIngombroArea_CCENTRALE + TCPParameter.Z + OffsetSicurezza.Avuoto THEN
						QuotaFuoriIngombro_Z_AVUOTO_CCENTRALE := AltezzaDiIngombroArea_CCENTRALE + TCPParameter.Z + OffsetSicurezza.Avuoto;
					END_IF
					IF QuotaFuoriIngombro_Z_ConPEZZO <= AltezzaDiIngombroArea_CCENTRALE + Dimensione_Z_ElementoInPresaX_Ingombro + OffsetSicurezza.ConPacco THEN//WorkArea^[a].Z + WorkArea^[a].H + Dimensione_Z_ElementoInPresaX_Ingombro + OFFSETSICUREZZA_Z THEN
						QuotaFuoriIngombro_Z_ConPEZZO := AltezzaDiIngombroArea_CCENTRALE + Dimensione_Z_ElementoInPresaX_Ingombro + OffsetSicurezza.ConPacco;//WorkArea^[a].Z + WorkArea^[a].H + Dimensione_Z_ElementoInPresaX_Ingombro + OFFSETSICUREZZA_Z;
					END_IF
				END_IF
			END_FOR
			
			(* Valuto I Pick-Point *)
			(*CASE TIPO_RIBALTINO OF
				RIBALTINO_DOPO_SQUADRO:
					FOR P:=1 TO MAXPICKPOINT DO
						AltezzaDiIngombroPuntiPrelievo := 0;
						IF  WorkPickPoint^[P].Zh + WorkPickPointState^[P].ZDim >= WorkPickPointDimension[P].Zdim THEN // Se Altezza orrizzontale Ribaltino + Zpacco >= Ingombro Verticale Ribaltino
							AltezzaDiIngombroPuntiPrelievo := WorkPickPoint^[P].Zh + WorkPickPointState^[P].ZDim;
						END_IF
						IF WorkPickPoint^[P].Zv + WorkPickPointState^[P].ZTilter + WorkPickPointState^[P].YDim >= WorkPickPointDimension[P].Zdim THEN // Se Altezza Vertivale Ribaltino + Quota Fermo + Ypacco >= Ingombro Verticale Ribaltino
							AltezzaDiIngombroPuntiPrelievo := WorkPickPoint^[P].Zv + WorkPickPointState^[P].ZTilter + WorkPickPointState^[P].YDim;
						END_IF
						IF WorkPickPointDimension[P].Zdim >= AltezzaDiIngombroPuntiPrelievo THEN //Se Ingombro Verticale Ribaltino >= Dell'ingombro valutato sopra
							AltezzaDiIngombroPuntiPrelievo := WorkPickPointDimension[P].Zdim;
						END_IF
						IF QuotaFuoriIngombro_Z_AVUOTO_CCENTRALE <= AltezzaDiIngombroPuntiPrelievo + TCPParameter.Z + OffsetSicurezza.Avuoto THEN //Se Quota fuori ingombro <= dell' ingombro del punto di prelievo
							QuotaFuoriIngombro_Z_AVUOTO_CCENTRALE := AltezzaDiIngombroPuntiPrelievo + TCPParameter.Z + OffsetSicurezza.Avuoto;
						END_IF				
					END_FOR
				RIBALTINO_DIRETTO :
					FOR P:=1 TO MAXPICKPOINT DO
						AltezzaDiIngombroPuntiPrelievo := 0;
						IF  WorkPickPoint^[P].Zh + WorkPickPointState^[P].ZDim >= WorkPickPointDimension[P].Zdim THEN // Se Altezza orrizzontale Ribaltino + Zpacco >= Ingombro Verticale Ribaltino
							AltezzaDiIngombroPuntiPrelievo := WorkPickPoint^[P].Zh + WorkPickPointState^[P].ZDim;
						END_IF
						IF WorkPickPoint^[P].Zv + WorkPickPointState^[P].ZTilter + WorkPickPointState^[P].XDim >= WorkPickPointDimension[P].Zdim THEN // Se Altezza Vertivale Ribaltino + Quota Fermo + Ypacco >= Ingombro Verticale Ribaltino
							AltezzaDiIngombroPuntiPrelievo := WorkPickPoint^[P].Zv + WorkPickPointState^[P].ZTilter + WorkPickPointState^[P].XDim;
						END_IF
						IF WorkPickPointDimension[P].Zdim >= AltezzaDiIngombroPuntiPrelievo THEN //Se Ingombro Verticale Ribaltino >= Dell'ingombro valutato sopra
							AltezzaDiIngombroPuntiPrelievo := WorkPickPointDimension[P].Zdim;
						END_IF
						IF QuotaFuoriIngombro_Z_AVUOTO_CCENTRALE <= AltezzaDiIngombroPuntiPrelievo + TCPParameter.Z + OffsetSicurezza.Avuoto THEN //Se Quota fuori ingombro <= dell' ingombro del punto di prelievo
							QuotaFuoriIngombro_Z_AVUOTO_CCENTRALE := AltezzaDiIngombroPuntiPrelievo + TCPParameter.Z + OffsetSicurezza.Avuoto;
						END_IF				
					END_FOR
			END_CASE*)
			
			END_IF //riferito all'IF dello stato della missione	
	
	WAMANAGER_CICLO_PRELIEVO_PACCO_END,
		
	WAMANAGER_CICLO_DEPOSITO_PACCO_RUN:
		IF Mission^.State = MISSION_STATE_NOP OR Mission^.State = MISSION_STATE_PRELIEVO_PACCO_END THEN
			//QuotaX_ConsensoRotazionePinza_Raggiunta := FALSE;
			QuotaFuoriIngombro_Z_AVUOTO_CCENTRALE := 0;
			QuotaFuoriIngombro_Z_ConPEZZO := 0;
			(* Valuto gli ostacoli per calcolare il fuori ingombro di Z *)
			//IF Mission^.JPickVO = 0 THEN
			//	OffsetSicurezzaConPacco := OffsetSicurezza.ConPacco;
		//	ELSE
		//		OffsetSicurezzaConPacco := OffsetSicurezza.ConPacco + 200;
		//	END_IF
			
			FOR f:=1 TO MAXFOOTPRINT DO	
				IF QuotaFuoriIngombro_Z_AVUOTO_CCENTRALE <= WorkFootPrint^[f].Z + WorkFootPrint^[f].ZDim + TCPParameter.Z + OffsetSicurezza.Avuoto THEN
					QuotaFuoriIngombro_Z_AVUOTO_CCENTRALE := WorkFootPrint^[f].Z + WorkFootPrint^[f].ZDim + TCPParameter.Z + OffsetSicurezza.Avuoto;
				END_IF
				IF Mission^.TPick = TPICK_PACK THEN
					IF QuotaFuoriIngombro_Z_ConPEZZO <= WorkFootPrint^[f].Z + WorkFootPrint^[f].ZDim + Dimensione_Z_ElementoInPresaX_Ingombro + OffsetSicurezzaConPacco THEN
						QuotaFuoriIngombro_Z_ConPEZZO := WorkFootPrint^[f].Z + WorkFootPrint^[f].ZDim + Dimensione_Z_ElementoInPresaX_Ingombro + OffsetSicurezzaConPacco;
					END_IF
				END_IF
			END_FOR
			(* Valuto le aree *)
			FOR a:=1 TO MAXAREA DO
				AltezzaDiIngombroArea_CCENTRALE := 0;
				IF WorkArea^[a].Typology <> TYPOLOGY_LAYER AND  WorkArea^[a].Typology <> TYPOLOGY_STACK THEN
					IF WorkAreaState^[a].H > WorkAreaState^[a].HPL THEN
						AltezzaDiIngombroArea_CCENTRALE := WorkAreaState^[a].H;
					ELSE
						AltezzaDiIngombroArea_CCENTRALE := WorkAreaState^[a].HPL;
					END_IF
					IF QuotaFuoriIngombro_Z_AVUOTO_CCENTRALE <= AltezzaDiIngombroArea_CCENTRALE + TCPParameter.Z + OffsetSicurezza.Avuoto THEN
						QuotaFuoriIngombro_Z_AVUOTO_CCENTRALE := AltezzaDiIngombroArea_CCENTRALE + TCPParameter.Z + OffsetSicurezza.Avuoto;
					END_IF
					IF QuotaFuoriIngombro_Z_ConPEZZO <=  AltezzaDiIngombroArea_CCENTRALE + Dimensione_Z_ElementoInPresaX_Ingombro + OffsetSicurezzaConPacco THEN
						QuotaFuoriIngombro_Z_ConPEZZO :=  AltezzaDiIngombroArea_CCENTRALE + Dimensione_Z_ElementoInPresaX_Ingombro + OffsetSicurezzaConPacco;
					END_IF
				end_if
			END_FOR
			
			(* Valuto I Pick-Point *)
			(*CASE TIPO_RIBALTINO OF
				RIBALTINO_DOPO_SQUADRO:
					FOR P:=1 TO MAXPICKPOINT DO
						AltezzaDiIngombroPuntiPrelievo := 0;
						IF  WorkPickPoint^[P].Zh + WorkPickPointState^[P].ZDim >= WorkPickPointDimension[P].Zdim THEN // Se Altezza orrizzontale Ribaltino + Zpacco >= Ingombro Verticale Ribaltino
							AltezzaDiIngombroPuntiPrelievo := WorkPickPoint^[P].Zh + WorkPickPointState^[P].ZDim;
						END_IF
						IF WorkPickPoint^[P].Zv + WorkPickPointState^[P].ZTilter + WorkPickPointState^[P].YDim >= WorkPickPointDimension[P].Zdim THEN // Se Altezza Vertivale Ribaltino + Quota Fermo + Ypacco >= Ingombro Verticale Ribaltino
							AltezzaDiIngombroPuntiPrelievo := WorkPickPoint^[P].Zv + WorkPickPointState^[P].ZTilter + WorkPickPointState^[P].YDim;
						END_IF
						IF WorkPickPointDimension[P].Zdim >= AltezzaDiIngombroPuntiPrelievo THEN //Se Ingombro Verticale Ribaltino >= Dell'ingombro valutato sopra
							AltezzaDiIngombroPuntiPrelievo := WorkPickPointDimension[P].Zdim;
						END_IF
						IF QuotaFuoriIngombro_Z_AVUOTO_CCENTRALE <= AltezzaDiIngombroPuntiPrelievo + TCPParameter.Z + OffsetSicurezza.Avuoto THEN //Se Quota fuori ingombro <= dell' ingombro del punto di prelievo
							QuotaFuoriIngombro_Z_AVUOTO_CCENTRALE := AltezzaDiIngombroPuntiPrelievo + TCPParameter.Z + OffsetSicurezza.Avuoto;
						END_IF				
					END_FOR
				RIBALTINO_DIRETTO :
					FOR P:=1 TO MAXPICKPOINT DO
						AltezzaDiIngombroPuntiPrelievo := 0;
						IF  WorkPickPoint^[P].Zh + WorkPickPointState^[P].ZDim >= WorkPickPointDimension[P].Zdim THEN // Se Altezza orrizzontale Ribaltino + Zpacco >= Ingombro Verticale Ribaltino
							AltezzaDiIngombroPuntiPrelievo := WorkPickPoint^[P].Zh + WorkPickPointState^[P].ZDim;
						END_IF
						IF WorkPickPoint^[P].Zv + WorkPickPointState^[P].ZTilter + WorkPickPointState^[P].XDim >= WorkPickPointDimension[P].Zdim THEN // Se Altezza Vertivale Ribaltino + Quota Fermo + Ypacco >= Ingombro Verticale Ribaltino
							AltezzaDiIngombroPuntiPrelievo := WorkPickPoint^[P].Zv + WorkPickPointState^[P].ZTilter + WorkPickPointState^[P].XDim;
						END_IF
						IF WorkPickPointDimension[P].Zdim >= AltezzaDiIngombroPuntiPrelievo THEN //Se Ingombro Verticale Ribaltino >= Dell'ingombro valutato sopra
							AltezzaDiIngombroPuntiPrelievo := WorkPickPointDimension[P].Zdim;
						END_IF
						IF QuotaFuoriIngombro_Z_AVUOTO_CCENTRALE <= AltezzaDiIngombroPuntiPrelievo + TCPParameter.Z + OffsetSicurezza.Avuoto THEN //Se Quota fuori ingombro <= dell' ingombro del punto di prelievo
							QuotaFuoriIngombro_Z_AVUOTO_CCENTRALE := AltezzaDiIngombroPuntiPrelievo + TCPParameter.Z + OffsetSicurezza.Avuoto;
						END_IF				
					END_FOR
			END_CASE
			*)
		END_IF //riferito all'IF dello stato della missione	
		*)
		(* Controllo della posizione X per dare OK alla rotazione della pinza per evitare che vada a sbattere *)
	(*	IF QuotaFuoriIngombro_Z_ConPEZZO >= (AltezzaDaPavimentoAPiastraSupportoColonnaCentrale - AltezzaPinzaDaTastatoreAFlangiaMotore - 100) AND 
			(ModuleAX_X^.Ax^.Status.ActPosition - (Dimensioni_Pinza.Lunghezza / 2) >= Quota_X_CentroColonnaCentrale + LarghezzaPiastraSupportoColonnaCentrale/2 + 50) OR 
			(ModuleAX_X^.Ax^.Status.ActPosition + (Dimensioni_Pinza.Lunghezza / 2) <= Quota_X_CentroColonnaCentrale - LarghezzaPiastraSupportoColonnaCentrale/2 - 50) THEN
			QuotaX_ConsensoRotazionePinza_Raggiunta := TRUE;
		END_IF*)
		
	//WAMANAGER_CICLO_DEPOSITO_PACCO_END;
	
END_CASE

(*
(* Punto di approccio iniziale - Necessario per lo start lenta *)
IF Mission^.TPick = TPICK_PALLET OR Mission^.TPick = TPICK_LAYER THEN
	Traiettoria^.PuntoDiApproccioStartPoint.X := Mission^.XPick;
	Traiettoria^.PuntoDiApproccioStartPoint.Y := Mission^.YPick;
	IF Mission^.TPick = TPICK_LAYER AND 						// SE il tipo di prelievo è PRELIEVO FALDA
		WorkArea^[Mission^.PPick].DoLearn_Z = 1 THEN					//se è necessario effettuare l'apprendimento
		Traiettoria^.PuntoDiApproccioStartPoint.Z := WorkArea^[Mission^.PPick].Learn_Z  + OffsetPrelieviLenti.Falde;	// La quota di start lenta verticale coincide con la quota assegnata alla WorkArea come quota di start apprendimento
	ELSIF Mission^.TPick = TPICK_LAYER AND 						// SE il tipo di prelievo è PRELIEVO FALDA
		WorkArea^[Mission^.PPick].DoLearn_Z = 2 THEN					//se NON DEVO effettuare l'apprendimento
		Traiettoria^.PuntoDiApproccioStartPoint.Z := WorkArea^[Mission^.PPick].Learned_Z + OffsetPrelieviLenti.Falde;//WorkArea^[Mission^.PPick].Z + WorkArea^[Mission^.PPick].H + OFFSETLENTAZ;	// La quota di start lenta verticale coincide con l'altezza della WA + altezza reale + offset.. vado piano da questa quota fino al tocco dei tastatori
	ELSIF Mission^.TPick = TPICK_PALLET AND 					// SE il tipo di prelievo è PRELIEVO FALDA
		WorkArea^[Mission^.PPick].DoLearn_Z = 1 THEN					//se è necessario effettuare l'apprendimento
		Traiettoria^.PuntoDiApproccioStartPoint.Z := WorkArea^[Mission^.PPick].Learn_Z + OffsetPrelieviLenti.Pallet;	// La quota di start lenta verticale coincide con la quota assegnata alla WorkArea come quota di start apprendimento
	ELSIF Mission^.TPick = TPICK_PALLET AND 					// SE il tipo di prelievo è PRELIEVO FALDA
		WorkArea^[Mission^.PPick].DoLearn_Z = 2 THEN					//se è necessario effettuare l'apprendimento
		Traiettoria^.PuntoDiApproccioStartPoint.Z := WorkArea^[Mission^.PPick].Learned_Z + OffsetPrelieviLenti.Pallet;	// La quota di start lenta verticale coincide con la quota assegnata alla WorkArea come quota di start apprendimento
	ELSE																				// Altrimenti, la quota di prelievo equivale alla quota di Prelievo + Offset 
		Traiettoria^.PuntoDiApproccioStartPoint.Z := Mission^.ZPick + OffsetPrelieviLenti.Pacco;
	END_IF
	Traiettoria^.PuntoDiApproccioStartPoint.K := Mission^.KPick;
	Traiettoria^.PuntoDiApproccioStartPoint.J := Mission^.JPick;
ELSE
	Traiettoria^.PuntoDiApproccioStartPoint.X := Mission^.XPick;
	Traiettoria^.PuntoDiApproccioStartPoint.Y := Mission^.YPick;
	Traiettoria^.PuntoDiApproccioStartPoint.Z := Mission^.ZPick;
	Traiettoria^.PuntoDiApproccioStartPoint.K := Mission^.KPick;
	Traiettoria^.PuntoDiApproccioStartPoint.J := Mission^.JPick;
END_IF
*)

///////////////////////////////////////////////////////////////////////////////////////////////////////////////////////////////////////////////////////////
///////////////////////////////////////////////////////////////////////////////////////////////////////////////////////////////////////////////////////////

(* Punto iniziale - Cincidente con il punto di prelievo *)
Traiettoria^.StartPoint.X := Mission^.XPick;
Traiettoria^.StartPoint.Y := Mission^.YPick;
Traiettoria^.StartPoint.Z := Mission^.ZPick;
Traiettoria^.StartPoint.K := Mission^.KPick;
Traiettoria^.StartPoint.J := Mission^.JPick;

///////////////////////////////////////////////////////////////////////////////////////////////////////////////////////////////////////////////////////////
///////////////////////////////////////////////////////////////////////////////////////////////////////////////////////////////////////////////////////////
(* Punto intermedio 1 - E' il punto avente coordinata Z maggiore della coordinata di partenza e tutte le altre coordinate sono uguali *)
Traiettoria^.PuntoIntermedio[1].X := Mission^.XPick;
Traiettoria^.PuntoIntermedio[1].Y := Mission^.YPick;
IF Mission^.TPick = TPICK_PACK THEN
	Traiettoria^.PuntoIntermedio[1].Z := QuotaFuoriIngombro_Z_ConPEZZO;	
ELSIF Mission^.TPick = TPICK_LAYER THEN	
	Traiettoria^.PuntoIntermedio[1].Z := QuotaFuoriIngombro_Z_ConFALDA;	
ELSIF Mission^.TPick = TPICK_PALLET THEN
	Traiettoria^.PuntoIntermedio[1].Z := QuotaFuoriIngombro_Z_ConPALLET;
END_IF		
Traiettoria^.PuntoIntermedio[1].K := Mission^.KPick;
Traiettoria^.PuntoIntermedio[1].J := Mission^.JPick;

///////////////////////////////////////////////////////////////////////////////////////////////////////////////////////////////////////////////////////////
///////////////////////////////////////////////////////////////////////////////////////////////////////////////////////////////////////////////////////////
(* Punto intermedio 2 - E' il punto avente coordinata Z uguale a quella del punto 1, coordinata X,Y,J e K uguale a quella del punto di approccio *)
Traiettoria^.PuntoIntermedio[2].X := Mission^.XPlaceApproach;
Traiettoria^.PuntoIntermedio[2].Y := Mission^.YPlaceApproach;
Traiettoria^.PuntoIntermedio[2].Z := Traiettoria^.PuntoIntermedio[1].Z;
Traiettoria^.PuntoIntermedio[2].K := Mission^.KPick;
Traiettoria^.PuntoIntermedio[2].J := Mission^.JPlaceApproach;

///////////////////////////////////////////////////////////////////////////////////////////////////////////////////////////////////////////////////////////
///////////////////////////////////////////////////////////////////////////////////////////////////////////////////////////////////////////////////////////
(* Punto di approccio finale :
- nel caso di deposito falda su catasta con apprendimento, la quota Z di approccio coincide con la quota di start lenta
- nel caso di deposito falda su catasta SENZA apprendimento, la quota Z di approccio coincide con la quota di start lenta per evitare che se c'è un pallet fuori sagoma, evitiamo collisioni brusche della pinza*)

Traiettoria^.PuntoDiApproccioEndPoint.X := Mission^.XPlaceApproach;
Traiettoria^.PuntoDiApproccioEndPoint.Y := Mission^.YPlaceApproach;
(*
IF Mission^.TPick = TPICK_LAYER AND 						// se ho tipo di prelievo falda
(WorkArea^[Mission^.PPlace].Typology = TYPOLOGY_STACK AND 	// e se è tipo di deposito su catasta vuoti
WorkArea^[Mission^.PPlace].DoLearn_Z = 1)  THEN					// e se è necessario effettuare l'apprendimento sulla catasta vuoti
	Traiettoria^.PuntoDiApproccioEndPoint.Z := WorkArea^[Mission^.PPlace].Learn_Z;	// La quota di start lenta verticale coincide con la quota assegnata alla WorkArea come quota di start apprendimento
	Quota_Attesa_Caduta_Falda_Z := WorkArea^[Mission^.PPick].Learned_Z + OffsetCadutaFalda;
ELSIF Mission^.TPick = TPICK_LAYER AND 						// se ho tipo di prelievo falda
(WorkArea^[Mission^.PPlace].Typology = TYPOLOGY_STACK AND 	// e se è tipo di deposito su catasta vuoti
WorkArea^[Mission^.PPlace].DoLearn_Z = 2)  THEN					// e se NON è necessario effettuare l'apprendimento sulla catasta vuoti
	Traiettoria^.PuntoDiApproccioEndPoint.Z := WorkArea^[Mission^.PPlace].Learned_Z + OffsetPrelieviLenti.Pallet;	// La quota di start lenta verticale coincide con la quota assegnata alla WorkArea come quota di start apprendimento
	Quota_Attesa_Caduta_Falda_Z := WorkArea^[Mission^.PPick].Learned_Z + OffsetCadutaFalda;
ELSE																				// Altrimenti,(caso di deposito pacco o falda su piazzola: la quota di DEPOSITO equivale alla quota di inizo approccio 
	Traiettoria^.PuntoDiApproccioEndPoint.Z := Mission^.ZPlaceApproach;
	Quota_Attesa_Caduta_Falda_Z := WorkArea^[Mission^.PPick].Learned_Z + OffsetCadutaFalda;
END_IF
*)
Traiettoria^.PuntoDiApproccioEndPoint.J := Mission^.JPlaceApproach;
Traiettoria^.PuntoDiApproccioEndPoint.K := Mission^.KPick;

/////////////////////////////////////////////////////////////////////////////////////////////////////////////////////////////////////////////////////////////
/////////////////////////////////////////////////////////////////////////////////////////////////////////////////////////////////////////////////////////////
(* Punto finale*)
Traiettoria^.EndPoint.X := Mission^.XPlace;
Traiettoria^.EndPoint.Y := Mission^.YPlace;
Traiettoria^.EndPoint.Z := Mission^.ZPlace;
Traiettoria^.EndPoint.K := Mission^.KPlace;
Traiettoria^.EndPoint.J := Mission^.JPlace;

(* Setto la quota minima di fuori ingombro che mi permette di star fuori dal filo delle barriere orrizontali *)
IF QuotaFuoriIngombro_Z_AVUOTO_CCENTRALE < 1450 THEN
	QuotaFuoriIngombro_Z_AVUOTO_CCENTRALE := 1450;
END_IF

Traiettoria^.PassModeGlobalEnable := AbilitazionePassModeGlobale;

END_FUNCTION_BLOCK

// ---- POUs/TFPalletizerDataTF/Utility Varie/TFCalcolaFuoriIngombroY_oo.TcPOU
FUNCTION_BLOCK TFCalcolaFuoriIngombroY_oo
VAR_INPUT
	
	WorkArea : POINTER TO TFMachinePalletizer_WorkArea;
	WorkAreaState : POINTER TO TFMachinePalletizer_WorkAreaState;
	Pallet : POINTER TO  TFMachinePalletizer_Pallet;
	ModuleAX_J : POINTER TO TFModulePalletizer_AxJ_Lastre;
	ModuleAX_Y : POINTER TO TFModulePalletizer_Ax;
	AngoloRotazioneDestinazionePinza : REAL;
END_VAR
VAR_OUTPUT
	Errore : TFError_WAM;
	QuotaFuoriIngombro_Y_Calcolata : LREAL;
END_VAR
VAR
	
END_VAR


QuotaFuoriIngombro_Y_Calcolata := 0;
(* Calcolo gli ingombri della pinza nelle varie direzioni *)
TFCalcoliIngombroPinza(Mission := Mission,
							WorkAreaManager := WorkAreaManager,
							ModuleAX_J := ModuleAX_J,
							AngoloRotazioneDestinazionePinza:= AngoloRotazioneDestinazionePinza,
							IngombroX_Pos := ADR(IngombroX_Pos),
							IngombroY_Pos := ADR(IngombroY_Pos),
							IngombroX_Neg := ADR(IngombroX_Neg),
							IngombroY_Neg := ADR(IngombroY_Neg),
							IngombroZ_Pos := ADR(IngombroZ_Pos),
							IngombroZ_Neg := ADR(IngombroZ_Neg),
							IngombroY_Tot := ADR(IngombroY_Tot),
							IngombroDestinazioneX_Pos := ADR(IngombroDestinazioneX_Pos),
							IngombroDestinazioneY_Pos := ADR(IngombroDestinazioneY_Pos),
							IngombroDestinazioneX_Neg := ADR(IngombroDestinazioneX_Neg),
							IngombroDestinazioneY_Neg := ADR(IngombroDestinazioneY_Neg),
							IngombroDestinazioneZ_Pos := ADR(IngombroDestinazioneZ_Pos),
							IngombroDestinazioneZ_Neg := ADR(IngombroDestinazioneZ_Neg),
							IngombroMaxX_Pos := ADR(IngombroMaxX_Pos),
							IngombroMaxY_Pos := ADR(IngombroMaxY_Pos),
							IngombroMaxX_Neg := ADR(IngombroMaxX_Neg),
							IngombroMaxY_Neg := ADR(IngombroMaxY_Neg),
							IngombroMaxZ_Pos := ADR(IngombroMaxZ_Pos),
							IngombroMaxZ_Neg := ADR(IngombroMaxZ_Neg));

CASE VERSO_PALLETTIZZATORE OF
	{region " Pallettizzatore DX "}					
	PALLETTIZZATORE_DX:
		CASE RIFERIMENTO_POSTAZIONE_WA OF
			{Region "ANGOLO DX" }
			ANGOLO_DX:
			
				IF AngoloRotazioneDestinazionePinza > 90 THEN					
				
					QuotaFuoriIngombro_Y_Calcolata := WorkArea^.Y + 					(* Quota Y Postazione *)																									
													WorkAreaState^.Supporto.YDim +(* Dimensione/2 del Pallet/Cassa/Cavallina *)
													OffsetSicurezza.Y.Avuoto;
										
				ELSIF AngoloRotazioneDestinazionePinza < 90 THEN
									
					QuotaFuoriIngombro_Y_Calcolata := WorkArea^.Y - 					(* Quota Y Postazione *)																									
													//WorkAreaState^.Supporto.YDim/2;(* Dimensione/2 del Pallet/Cassa/Cavallina *)
													OffsetSicurezza.Y.Avuoto;
				ELSE
					
					QuotaFuoriIngombro_Y_Calcolata := WorkArea^.Y;// + 					(* Quota Y Postazione *)																									
													//WorkAreaState^.Supporto.YDim +(* Dimensione/2 del Pallet/Cassa/Cavallina *)
													//OffsetSicurezza.Y.Avuoto;
				END_IF
			{endregion}
			{Region "CENTRALE" }
			CENTRALE :
			
				IF AngoloRotazioneDestinazionePinza > 90 THEN					
				
					QuotaFuoriIngombro_Y_Calcolata := WorkArea^.Y + 					(* Quota Y Postazione *)																									
													WorkAreaState^.Supporto.YDim/2 +(* Dimensione/2 del Pallet/Cassa/Cavallina *)
													OffsetSicurezza.Y.Avuoto;
										
				ELSIF AngoloRotazioneDestinazionePinza < 90 THEN
									
					QuotaFuoriIngombro_Y_Calcolata := WorkArea^.Y - 					(* Quota Y Postazione *)																									
													WorkAreaState^.Supporto.YDim/2 -(* Dimensione/2 del Pallet/Cassa/Cavallina *)
													OffsetSicurezza.Y.Avuoto;
				ELSE
					
					QuotaFuoriIngombro_Y_Calcolata := WorkArea^.Y;// + 					(* Quota Y Postazione *)																									
													//WorkAreaState^.Supporto.YDim +(* Dimensione/2 del Pallet/Cassa/Cavallina *)
													//OffsetSicurezza.Y.Avuoto;
				END_IF
			{endregion}
			{Region "ANGOLO SX" }
			ANGOLO_SX :
			
				IF AngoloRotazioneDestinazionePinza > 90 THEN					
				
					QuotaFuoriIngombro_Y_Calcolata := WorkArea^.Y + 					(* Quota Y Postazione *)																									
													WorkAreaState^.Supporto.YDim +(* Dimensione/2 del Pallet/Cassa/Cavallina *)
													OffsetSicurezza.Y.Avuoto;
										
				ELSIF AngoloRotazioneDestinazionePinza < 90 THEN
									
					QuotaFuoriIngombro_Y_Calcolata := WorkArea^.Y - 					(* Quota Y Postazione *)																									
													//WorkAreaState^.Supporto.YDim/2;(* Dimensione/2 del Pallet/Cassa/Cavallina *)
													OffsetSicurezza.Y.Avuoto;
				ELSE
					
					QuotaFuoriIngombro_Y_Calcolata := WorkArea^.Y;// + 					(* Quota Y Postazione *)																									
													//WorkAreaState^.Supporto.YDim +(* Dimensione/2 del Pallet/Cassa/Cavallina *)
													//OffsetSicurezza.Y.Avuoto;
				END_IF
			{endregion}

			{Region "XDX_YCENTRALE" }			
			XDX_YCENTRALE:	
			
				;		
			{endregion}

			{Region "XSX_YCENTRALE" }
			XSX_YCENTRALE:
			
				;
			{endregion}
			
		ELSE
			Errore.Code := ErrWAM_FTC_PostazioneNONDefinita;
		END_CASE	
	{endregion}	
	{region " Pallettizzatore SX "}	
	PALLETTIZZATORE_SX:

		CASE RIFERIMENTO_POSTAZIONE_WA OF
			{Region "ANGOLO DX" }
			ANGOLO_DX:
			
				IF AngoloRotazioneDestinazionePinza > 95 THEN					
				
					QuotaFuoriIngombro_Y_Calcolata := WorkArea^.Y + 					(* Quota Y Postazione *)																									
													WorkAreaState^.Supporto.YDim +(* Dimensione/2 del Pallet/Cassa/Cavallina *)
													IngombroDestinazioneY_Neg +
													OffsetSicurezza.Y.Avuoto;
										
				ELSIF AngoloRotazioneDestinazionePinza < 85 THEN
									
					QuotaFuoriIngombro_Y_Calcolata := WorkArea^.Y - 					(* Quota Y Postazione *)																									
													//WorkAreaState^.Supporto.YDim/2;(* Dimensione/2 del Pallet/Cassa/Cavallina *)
													IngombroDestinazioneY_Pos -
													OffsetSicurezza.Y.Avuoto;
				ELSE
					
					IF ModuleAX_Y^.Ax^.Status.ActPosition >= WorkArea^.Y THEN 
						QuotaFuoriIngombro_Y_Calcolata := WorkArea^.Y + 					(* Quota Y Postazione *)																									
															WorkAreaState^.Supporto.YDim +(* Dimensione/2 del Pallet/Cassa/Cavallina *)
															IngombroDestinazioneY_Neg +
															OffsetSicurezza.Y.Avuoto;
					ELSE
						QuotaFuoriIngombro_Y_Calcolata := WorkArea^.Y - 					(* Quota Y Postazione *)																									
															//WorkAreaState^.Supporto.YDim +(* Dimensione/2 del Pallet/Cassa/Cavallina *)
															IngombroDestinazioneY_Pos +
															OffsetSicurezza.Y.Avuoto;

					END_IF
				END_IF
			{endregion}
			{Region "CENTRALE" }				
			CENTRALE :
				IF AngoloRotazioneDestinazionePinza > 90 THEN					
				
					QuotaFuoriIngombro_Y_Calcolata := WorkArea^.Y + 					(* Quota Y Postazione *)																									
													WorkAreaState^.Supporto.YDim/2 +(* Dimensione/2 del Pallet/Cassa/Cavallina *)
													OffsetSicurezza.Y.Avuoto;
										
				ELSIF AngoloRotazioneDestinazionePinza < 90 THEN
									
					QuotaFuoriIngombro_Y_Calcolata := WorkArea^.Y - 					(* Quota Y Postazione *)																									
													WorkAreaState^.Supporto.YDim/2 -(* Dimensione/2 del Pallet/Cassa/Cavallina *)
													OffsetSicurezza.Y.Avuoto;
				ELSE
					
					QuotaFuoriIngombro_Y_Calcolata := WorkArea^.Y;// + 					(* Quota Y Postazione *)																									
													//WorkAreaState^.Supporto.YDim +(* Dimensione/2 del Pallet/Cassa/Cavallina *)
													//OffsetSicurezza.Y.Avuoto;
				END_IF
			{endregion}
			{Region "ANGOLO SX" }
			ANGOLO_SX :
				IF AngoloRotazioneDestinazionePinza > 90 THEN					
				
					QuotaFuoriIngombro_Y_Calcolata := WorkArea^.Y + 					(* Quota Y Postazione *)																									
													WorkAreaState^.Supporto.YDim +(* Dimensione/2 del Pallet/Cassa/Cavallina *)
													OffsetSicurezza.Y.Avuoto;
										
				ELSIF AngoloRotazioneDestinazionePinza < 90 THEN
									
					QuotaFuoriIngombro_Y_Calcolata := WorkArea^.Y - 					(* Quota Y Postazione *)																									
													//WorkAreaState^.Supporto.YDim/2;(* Dimensione/2 del Pallet/Cassa/Cavallina *)
													OffsetSicurezza.Y.Avuoto;
				ELSE
					
					QuotaFuoriIngombro_Y_Calcolata := WorkArea^.Y;// + 					(* Quota Y Postazione *)																									
													//WorkAreaState^.Supporto.YDim +(* Dimensione/2 del Pallet/Cassa/Cavallina *)
													//OffsetSicurezza.Y.Avuoto;
				END_IF
			{endregion}
			{Region "XDX_YCENTRALE" }
			XDX_YCENTRALE:
				;
			{endregion}
			{Region "XSX_YCENTRALE" }
			XSX_YCENTRALE:
				;
			{endregion}		
							
		ELSE
			Errore.Code := ErrWAM_FTC_PostazioneNONDefinita;
		END_CASE
	{endregion}	
	ELSE
		;	
END_CASE

END_FUNCTION_BLOCK

// ---- POUs/TFPalletizerDataTF/Utility Varie/TFInverterV1000.TcPOU
FUNCTION_BLOCK TFInverterV1000
VAR_INPUT
	OperationCommand : POINTER TO UINT; //Comandi V1000
	DriveStatus : POINTER TO UINT;//Stato del Drive
	
	Power 		: BOOL; // Abilitazione Asse
	Run 		: BOOL; // Run Asse
	Reverse 	: BOOL; // Comando Rotazione Indietro
	ResetAlarm  : BOOL; // Comando di reset allarmi
END_VAR
VAR_OUTPUT
	DriveRun 		: BOOL;//Drive in stato di RUN
	ReverseRunning 	: BOOL; //Comando di Reverse
	DriveReady 		: BOOL;//Drive Ready
	DriveAlarm 		: BOOL;//Drive in allarme
	DriveFault		: BOOL;//Drive in Fault
END_VAR
VAR
	MEMResetAlarm : BOOL;
END_VAR


//Stato inverter
DriveRun 		:= DriveStatus^.0;
ReverseRunning 	:= DriveStatus^.1;
DriveReady 		:= DriveStatus^.5;
DriveAlarm 		:= DriveStatus^.6;
DriveFault 		:= DriveStatus^.7;

//Comando Inverter
OperationCommand^.0 := FALSE;
OperationCommand^.1 := FALSE;
OperationCommand^.3 := FALSE;

IF DriveReady THEN//Se è tutto ok attendo che arrivi un comando di movimento
	OperationCommand^.0 := Power AND Run;
	OperationCommand^.1 := Power AND Run AND Reverse;
ELSIF (DriveAlarm OR DriveFault) THEN //Se il drive è in FAULT o IN ALLARME attendo il comando di RESET allarmi
	OperationCommand^.3 := ResetAlarm;
	MEMResetAlarm := TRUE;
END_IF	

IF MEMResetAlarm AND DriveReady THEN
	MEMResetAlarm := FALSE;
END_IF

END_FUNCTION_BLOCK

// ---- POUs/TFPalletizerData/NON_USATE/TFCheckPalletFull.TcPOU
FUNCTION TFCheckPalletFull : INT
VAR_INPUT
	WorkArea : POINTER TO ARRAY [1..MAXAREA] OF TFMachinePalletizer_WorkArea;
	WorkAreaState : POINTER TO ARRAY [1..MAXAREA] OF TFMachinePalletizer_WorkAreaState;
	//PX_WorkArea : ARRAY [1..MAXAREA] OF BOOL;
	WorkPickPointState : POINTER TO ARRAY [1..MAXPICKPOINT] OF TFMachinePalletizer_WorkPickPointState;
	Forming : POINTER TO ARRAY [1..MAXFORMING] OF TFMachinePalletizer_Forming;
END_VAR
VAR
	i : INT;
	k : INT;
END_VAR

TFCheckPalletFull := 0;
FOR k := 1 TO MAXPICKPOINT DO
	//IF WorkPickPointState^[k].State = 1 THEN
		FOR i:=1 TO MAXAREA DO	
			IF WorkArea^[i].Enable = 1 AND WorkArea^[i].Typology = TYPOLOGY_PALLET AND 
				WorkArea^[i].Code = 0  AND 
				//WorkAreaState^[i].State <= WORKAREA_STATE_OCCUPIED_WORKING AND 
				(Forming^[WorkAreaState^[i].F].PackXP[WorkAreaState^[i].P].Grip <> -1 OR 
				Forming^[WorkAreaState^[i].F].PackXN[WorkAreaState^[i].P].Grip <> -1) THEN
				RETURN;
			END_IF
		END_FOR
	//ELSE
	//	;//RETURN;	
	//END_IF	
END_FOR	
	
TFCheckPalletFull := 1;

END_FUNCTION

// ---- POUs/TFPalletizerData/NON_USATE/TFClearWorkAreaStack.TcPOU
FUNCTION TFClearWorkAreaStack : BOOL
VAR_INPUT
	WorkArea : POINTER TO ARRAY [1..MAXAREA] OF TFMachinePalletizer_WorkArea;
	WorkAreaState : POINTER TO ARRAY [1..MAXAREA] OF TFMachinePalletizer_WorkAreaState;
	k : UINT;
END_VAR
VAR
END_VAR

TFClearWorkAreaStack := FALSE;

WorkArea^[k].LGV_Req := 0;
//WorkArea^[k].H := 1000;
WorkArea^[k].HPL := 0;
WorkArea^[k].Taped := -1;
WorkArea^[k].DoLearn_Z := 1;
WorkArea^[k].LGV_GetIn_GetOut := -1;
WorkAreaState^[k].F := -1;
WorkAreaState^[k].P := -1;
//WorkAreaState^[k].L := -1;
//WorkAreaState^[k].PN := -1;
WorkAreaState^[k].State := WORKAREA_STATE_FREE_DISABLED;
WorkAreaState^[k].PackPointerModified := FALSE;
WorkAreaState^[k].PackPointer := -1;
TFClearWorkAreaStateSlab(WorkAreaState,k);
IF WorkArea^[k].Jolly = 1 THEN
	 WorkArea^[k].Code := 0;
END_IF

END_FUNCTION

// ---- POUs/TFPalletizerData/TFClearWorkAreaStateSlab.TcPOU
FUNCTION TFClearWorkAreaStateSlab : BOOL
VAR_INPUT
	WorkAreaState : POINTER TO ARRAY [1..MAXAREA] OF TFMachinePalletizer_WorkAreaState;
	k : UINT;
END_VAR
VAR
	i : uINT;
	j : UINT;
END_VAR

TFClearWorkAreaStateSlab := FALSE;

FOR i:=1 TO MAXFORMINGPACK DO
	FOR j:=1 TO MAXHANDLINGSTACK DO
		WorkAreaState^[k].Slab[j] := EmptySlab;
	END_FOR
END_FOR
TFClearWorkAreaStateSlab := TRUE;

END_FUNCTION

// ---- POUs/TFPalletizerData/NON_USATE/TFGetEnableCode.TcPOU
FUNCTION TFGetEnableCode : ARRAY [1..MAXFORMINGCODE*MAXFORMING] OF INT
VAR_INPUT
	Forming : POINTER TO ARRAY [1..MAXFORMING] OF TFMachinePalletizer_Forming;
END_VAR
VAR
	EnableCode : ARRAY [1..MAXFORMINGCODE*MAXFORMING] OF INT;
	pp : UINT;
	pf : UINT;
	c : INT;
	i : UINT;
END_VAR

FOR i:=1 TO MAXFORMINGCODE*MAXFORMING DO
	EnableCode[i]:= 0;
END_FOR
c:=1; 
(* Per Tutte le Formature Attive *)
FOR pf:=1 TO MAXFORMING DO
	IF Forming^[pf].Enable = 1 THEN
		(* Per tutti i codici di Pallettizzazione Validi *)
		FOR pp:=1 TO MAXFORMINGCODE DO
			IF Forming^[pf].Code[pp] > 0 THEN
				EnableCode[c] := Forming^[pf].Code[pp];
				c := c+1;
			END_IF
		END_FOR
	END_IF
END_FOR
TFGetEnableCode := EnableCode;

END_FUNCTION

// ---- POUs/TFPalletizerData/NON_USATE/TFGripperNearTilter.TcPOU
FUNCTION TFGripperNearTilter : BOOL
VAR_INPUT
	PickPoint : TFMachinePalletizer_WorkPickPoint;
	Radius : LREAL;
	Modules : POINTER TO TFMachinePalletizer_Modules;
	
END_VAR
VAR
	Distance : LREAL;
END_VAR

TFGripperNearTilter := FALSE;

Distance := SQRT(((Modules^.Robot.XAx^.AxRef^.NcToPlc.ActPos-PickPoint.Xh)*(Modules^.Robot.XAx^.AxRef^.NcToPlc.ActPos-PickPoint.Xh))+
					((Modules^.Robot.YAx^.AxRef^.NcToPlc.ActPos-PickPoint.Yh)*(Modules^.Robot.YAx^.AxRef^.NcToPlc.ActPos-PickPoint.Yh))+
					((Modules^.Robot.ZAx^.AxRef^.NcToPlc.ActPos-PickPoint.Zh)*(Modules^.Robot.ZAx^.AxRef^.NcToPlc.ActPos-PickPoint.Zh)));


IF Distance <= Radius THEN
	TFGripperNearTilter := TRUE;
END_IF

END_FUNCTION

// ---- POUs/TFPalletizerData/NON_USATE/TFLeastUsedCode.TcPOU
FUNCTION TFLeastUsedCode : INT
VAR_INPUT
	EnableCode : ARRAY [1..MAXFORMINGCODE*MAXFORMING] OF INT;
	UsedCode : POINTER TO ARRAY [1..MAXFORMINGCODE] OF INT;
END_VAR
VAR
	Code : INT;
	i : INT;
	j : INT;
	Counter : INT;
	MinCounter : INT;
END_VAR

TFLeastUsedCode := 0;
Code := 0;
MinCounter := MAXFORMINGCODE + 1;

FOR i:=1 TO MAXFORMINGCODE*MAXFORMING DO
	IF EnableCode[i] > 0 THEN
		Counter := 0;
		FOR j:=1 TO MAXFORMINGCODE DO
			IF UsedCode^[j] = EnableCode[i] THEN
				Counter := Counter + 1;
			END_IF
		END_FOR
		IF Counter < MinCounter THEN
			MinCounter := Counter;
			Code := EnableCode[i];
		END_IF 
	END_IF
END_FOR

TFLeastUsedCode := Code;

END_FUNCTION

// ---- POUs/TFPalletizerData/NON_USATE/TFMostUsedCode.TcPOU
FUNCTION TFMostUsedCode : INT
VAR_INPUT
	EnableCode : ARRAY [1..MAXFORMINGCODE*MAXFORMING] OF INT;
	UsedCode : POINTER TO ARRAY [1..MAXFORMINGCODE] OF INT;
END_VAR
VAR
	Code : INT;
	i : INT;
	j : INT;
	Counter : INT;
	MaxCounter : INT;
END_VAR

TFMostUsedCode := 0;
Code := 0;
MaxCounter := 0;

FOR i:=1 TO MAXFORMINGCODE*MAXFORMING DO
	IF EnableCode[i] > 0 THEN
		Counter := 0;
		FOR j:=1 TO MAXFORMINGCODE DO
			IF UsedCode^[j] = EnableCode[i] THEN
				Counter := Counter + 1;
			END_IF
		END_FOR
		IF Counter > MaxCounter THEN
			MaxCounter := Counter;
			Code := EnableCode[i];
		END_IF 
	END_IF
END_FOR

TFMostUsedCode := Code;

END_FUNCTION

// ---- POUs/TFPalletizerData/NON_USATE/TFNextCommandToTilter.TcPOU
FUNCTION TFNextCommandToTilter : INT
VAR_INPUT
	WorkArea : POINTER TO ARRAY [1..MAXAREA] OF TFMachinePalletizer_WorkArea;
	WorkAreaState : POINTER TO ARRAY [1..MAXAREA] OF TFMachinePalletizer_WorkAreaState;
	DistanceFromWAPointer : ARRAY [1..MAXAREA] OF TFMachinePalletizer_WorkAreaSort;
	Forming : POINTER TO ARRAY [1..MAXFORMING] OF TFMachinePalletizer_Forming;
	Mission : POINTER TO TFMachinePalletizer_Mission;
	NextCode : INT;
END_VAR
VAR
	i : INT;
END_VAR

TFNextCommandToTilter := -1;

FOR i:=1 TO MAXAREA DO
	IF WorkArea^[DistanceFromWAPointer[i].cwa].Code = NextCode THEN
		IF WorkArea^[DistanceFromWAPointer[i].cwa].Enable = 1 AND Forming^[WorkAreaState^[DistanceFromWAPointer[i].cwa].F].Enable = 1 AND 
			WorkAreaState^[DistanceFromWAPointer[i].cwa].State = WORKAREA_STATE_OCCUPIED_WORKING THEN
				IF DistanceFromWAPointer[i].cwa = Mission^.PPlace THEN
					TFNextCommandToTilter := Forming^[WorkAreaState^[DistanceFromWAPointer[i].cwa].F].PackXP[WorkAreaState^[DistanceFromWAPointer[i].cwa].P + 1].Grip;
					RETURN;
				ELSE
					TFNextCommandToTilter := Forming^[WorkAreaState^[DistanceFromWAPointer[i].cwa].F].PackXP[WorkAreaState^[DistanceFromWAPointer[i].cwa].P].Grip;
					RETURN;
				END_IF	
		END_IF
	END_IF
END_FOR

END_FUNCTION

// ---- POUs/TFPalletizerData/NON_USATE/TFPackCodeOnWPP.TcPOU
FUNCTION TFPackCodeOnWPP : INT
VAR_INPUT
	WorkArea : POINTER TO ARRAY [1..MAXAREA] OF TFMachinePalletizer_WorkArea;
	WorkAreaState : POINTER TO ARRAY [1..MAXAREA] OF TFMachinePalletizer_WorkAreaState;
	WorkPickPointState : POINTER TO ARRAY [1..MAXPICKPOINT] OF TFMachinePalletizer_WorkPickPointState;
	Forming : POINTER TO ARRAY [1..MAXFORMING] OF TFMachinePalletizer_Forming;
END_VAR
VAR
	wpp : INT;
	i : INT;
	CodeAssignedToWA : BOOL; // TRUE se i codice è assegnato ad almeno una WA
END_VAR

TFPackCodeOnWPP := -1; 
CodeAssignedToWA := FALSE;

FOR wpp:=1 TO MAXPICKPOINT DO
	(* Verifico disponibilità Pacco *)
	IF WorkPickPointState^[wpp].State = WORKPICKPOINT_PRODOTTO_PRESENTE THEN
		(* Verifico se il codice è assegnato a qualche workarea e se la formatura è attiva *)
		FOR i:=1 TO MAXAREA DO
			IF WorkPickPointState^[wpp].Code = WorkArea^[wpp].Code THEN
				CodeAssignedToWA := TRUE;
				IF WorkArea^[wpp].Enable = 1 AND NOT Forming^[WorkAreaState^[wpp].F].Enable = 1 THEN
					TFPackCodeOnWPP := 1;//codice assegnato a workarea con formatura disabilitata
					RETURN;
				ELSIF NOT WorkArea^[wpp].Enable = 1 AND Forming^[WorkAreaState^[wpp].F].Enable = 1 THEN
					TFPackCodeOnWPP := 2;//codice assegnato a workarea disabilitata
					RETURN;
				ELSIF NOT WorkArea^[wpp].Enable = 1 AND NOT Forming^[WorkAreaState^[wpp].F].Enable = 1 THEN
					TFPackCodeOnWPP := 3;//codice assegnato a workarea disabilitata e con formatura disabilitata
					RETURN;
				END_IF	
			END_IF
		END_FOR	
		IF CodeAssignedToWA THEN
			TFPackCodeOnWPP := -1;
			RETURN;
		END_IF
	END_IF
	TFPackCodeOnWPP := 4; // Codice pacco non assegnato a nessuna workarea
END_FOR

END_FUNCTION

// ---- POUs/TFPalletizerData/NON_USATE/TFPackCodePresentToJollyWorkArea.TcPOU
FUNCTION TFPackCodePresentToJollyWorkArea : INT
VAR_INPUT
	HandlingPackTable : POINTER TO TFHandlingPackTable;
	WorkArea : POINTER TO ARRAY [1..MAXAREA] OF TFMachinePalletizer_WorkArea;
	WorkAreaState : POINTER TO ARRAY [1..MAXAREA] OF TFMachinePalletizer_WorkAreaState;
END_VAR
VAR
	w : INT;
	wa : INT;
	i : INT;
END_VAR

TFPackCodePresentToJollyWorkArea := 0; 

FOR w:=MAXHANDLINGPACK TO 1 BY -1 DO
	IF HandlingPackTable^.Table[w,1].PC > 0 THEN
		FOR wa:=1 TO MAXAREA DO
			IF WorkArea^[wa].Code = HandlingPackTable^.Table[w,1].PC THEN
				(* Verifico se la piazzola è in lavorazione *)
				(* Se è in lavorazione allora è inutile assegnarne un'altra con lo stesso codice *)
				IF WorkAreaState^[wa].State < WORKAREA_STATE_OCCUPIED_WORKED THEN
					TFPackCodePresentToJollyWorkArea := 0;
					RETURN;
				//ELSE
					//TFPackCodePresentToJollyWorkArea := WorkPickPointState^[w].Code;
				END_IF
				//RETURN;
			END_IF
		END_FOR
		TFPackCodePresentToJollyWorkArea := HandlingPackTable^.Table[w,1].PC;
	END_IF	
END_FOR

END_FUNCTION

// ---- POUs/TFPalletizerData/NON_USATE/TFPackCodePresentToZone.TcPOU
FUNCTION TFPackCodePresentToZone : INT
VAR_INPUT
	HandlingPackTable : POINTER TO TFHandlingPackTable;
	WorkAreaZone : POINTER TO TFMachinePalletizer_WorkAreaZone;
	WorkArea : INT;
END_VAR
VAR
	w : INT;
	n : INT;
	i : INT;
	a : INT;
END_VAR

TFPackCodePresentToZone := 0; 

FOR w:=MAXHANDLINGPACK TO 1 BY -1 DO
	IF HandlingPackTable^.Table[w,1].PC > 0 THEN
		FOR n:=1 TO MAXZONE DO
			FOR a:=1 TO MAXAREA DO
				IF WorkAreaZone^.Zone[n].WorkArea[a] = WorkArea THEN
					FOR i:=1 TO MAXFORMINGCODE DO
						(* Verifico se il Pacco presente nel WPP è destinato ad una Zona *)
						IF WorkAreaZone^.Zone[n].Code[i] = HandlingPackTable^.Table[w,1].PC THEN
							TFPackCodePresentToZone := HandlingPackTable^.Table[w,1].PC;
							RETURN;
						END_IF
					END_FOR
				END_IF
			END_FOR
		END_FOR
	END_IF
END_FOR

END_FUNCTION

// ---- POUs/TFPalletizerData/NON_USATE/TFPackOnPickPoint.TcPOU
FUNCTION TFPackOnPickPoint : BOOL
VAR_INPUT
	WorkPickPointState : POINTER TO ARRAY [1..MAXPICKPOINT] OF TFMachinePalletizer_WorkPickPointState;
END_VAR
VAR
	wpp : INT;
END_VAR

TFPackOnPickPoint := FALSE;

FOR wpp:=1 TO MAXPICKPOINT DO
	(* Verifico disponibilità Pacco *)
	IF WorkPickPointState^[wpp].State = WORKPICKPOINT_PRODOTTO_PRESENTE THEN
		TFPackOnPickPoint := TRUE;
	END_IF
END_FOR

END_FUNCTION

// ---- POUs/TFPalletizerData/NON_USATE/TFPalletizerCheckPalletLayerCode.TcPOU
FUNCTION TFPalletizerCheckPalletLayerCode : UINT
VAR_INPUT
	WorkArea : POINTER TO ARRAY [1..MAXAREA] OF TFMachinePalletizer_WorkArea;
	WorkAreaState : POINTER TO ARRAY [1..MAXAREA] OF TFMachinePalletizer_WorkAreaState;
	Forming : POINTER TO ARRAY [1..MAXFORMING] OF TFMachinePalletizer_Forming;
END_VAR
VAR
	f : UINT;
	i : UINT;
	PalletFound : BOOL;
	LayerFound : BOOL;
END_VAR

(* Verifica che la catasta pallett e la catasta vuoti abbiano codice uguale a quello della formatura attiva per del pacco presente nel punto di prelievo *)
TFPalletizerCheckPalletLayerCode := 0; 
PalletFound := FALSE;
LayerFound := FALSE;

FOR f:=1 TO MAXFORMING DO 
	(* Verifico Formature attive *)
	IF Forming^[f].Enable = 1 THEN
		(* Verifico se i codici Layer e Pallet sono presenti tra le WorkArea *)
		FOR i:=1 TO MAXAREA DO
			IF  WorkArea^[i].Typology = TYPOLOGY_STACK AND WorkArea^[i].Enable = 1 (*AND WorkAreaState^[i].State >= WORKAREA_STATE_OCCUPIED_WORKING*) THEN 
				IF WorkArea^[i].Pallet = Forming^[f].Pallet THEN
					PalletFound := TRUE; 
				END_IF	
			END_IF	
			IF  ((WorkArea^[i].Typology = TYPOLOGY_LAYER AND WorkArea^[i].Enable = 1  (*AND WorkAreaState^[i].State >= WORKAREA_STATE_OCCUPIED_WORKING*)) OR Forming^[f].Layer = 0) THEN 
				IF WorkArea^[i].Layer = Forming^[f].Layer or Forming^[f].Layer=0 THEN
					LayerFound := TRUE; 
				END_IF	
			END_IF	
		END_FOR	
		IF NOT PalletFound  THEN 
			TFPalletizerCheckPalletLayerCode := ErrPALLETCODENOTFOUND;
			RETURN; 
		ELSIF NOT LayerFound THEN	
			TFPalletizerCheckPalletLayerCode := ErrLAYERCODENOTFOUND;
			RETURN; 
		END_IF
	END_IF
END_FOR

END_FUNCTION

// ---- POUs/TFPalletizerData/NON_USATE/TFPalletizerPackValidation.TcPOU
FUNCTION TFPalletizerPackValidation : INT
VAR_INPUT
	WorkArea : POINTER TO ARRAY [1..MAXAREA] OF TFMachinePalletizer_WorkArea;
	WorkAreaState : POINTER TO ARRAY [1..MAXAREA] OF TFMachinePalletizer_WorkAreaState;
	WorkPickPointState : POINTER TO ARRAY [1..MAXPICKPOINT] OF TFMachinePalletizer_WorkPickPointState;
	Forming : POINTER TO ARRAY [1..MAXFORMING] OF TFMachinePalletizer_Forming;
	Mission : POINTER TO TFMachinePalletizer_Mission;
	AxisPar : POINTER TO Ax_Palletizer_Parameters;
END_VAR
VAR
	wpp : INT;
	i : INT;
	PackOffset : REAL;
	CodeAssignedToWA : BOOL; // TRUE se i codice è assegnato ad almeno una WA
	fcode : INT;
END_VAR

TFPalletizerPackValidation := 0; 
PackOffset := 50.0;

IF  Mission^.KPick >= AxisPar^.MaxPosition OR Mission^.KPick <= AxisPar^.MinPosition// OR
	(*Mission^.KPlace > AxisPar^.K.MaxPosition OR Mission^.KPlace < AxisPar^.K.MinPosition*) THEN
		TFPalletizerPackValidation := ErrCONFIGURAZIONEPINZASABGLIATA; // Configurazione Pinza non adatta al prelievo o al deposito
		RETURN;	
END_IF

FOR wpp:=1 TO MAXPICKPOINT DO
	(* Verifico disponibilità Pacco *)
	IF WorkPickPointState^[wpp].State = WORKPICKPOINT_PRODOTTO_PRESENTE THEN
		fcode := TFPalletizerGetFormingFromCode(Forming,WorkPickPointState^[wpp].Code);
		CASE TIPO_RIBALTINO OF
			RIBALTINO_DOPO_SQUADRO:
				IF fcode = 0 THEN
					TFPalletizerPackValidation := ErrPACKCODENOTVALID; // Codice non associato a formatura
					RETURN;			
				ELSIF (WorkPickPointState^[wpp].XDim < Forming^[fcode].PX - PackOffset OR
					WorkPickPointState^[wpp].XDim > Forming^[fcode].PX + PackOffset) OR
					(WorkPickPointState^[wpp].YDim < Forming^[fcode].PY - PackOffset  OR
					WorkPickPointState^[wpp].YDim > Forming^[fcode].PY + PackOffset) OR
					(WorkPickPointState^[wpp].ZDim < Forming^[fcode].PZ - PackOffset OR
					WorkPickPointState^[wpp].ZDim > Forming^[fcode].PZ + PackOffset)THEN
						TFPalletizerPackValidation := ErrPACKDIMENSIONNOTVALID; // Grandezze pacco errate
						RETURN;
				END_IF

			RIBALTINO_DIRETTO:
				IF fcode = 0 THEN
					TFPalletizerPackValidation := ErrPACKCODENOTVALID; // Codice non associato a formatura
					RETURN;			
				ELSIF (WorkPickPointState^[wpp].XDim < Forming^[fcode].PY - PackOffset OR
					WorkPickPointState^[wpp].XDim > Forming^[fcode].PY + PackOffset) OR
					(WorkPickPointState^[wpp].YDim < Forming^[fcode].PX - PackOffset  OR
					WorkPickPointState^[wpp].YDim > Forming^[fcode].PX + PackOffset) OR
					(WorkPickPointState^[wpp].ZDim < Forming^[fcode].PZ - PackOffset OR
					WorkPickPointState^[wpp].ZDim > Forming^[fcode].PZ + PackOffset)THEN
						TFPalletizerPackValidation := ErrPACKDIMENSIONNOTVALID; // Grandezze pacco errate
						RETURN;
				END_IF	
		END_CASE
		
	END_IF
END_FOR	

(*FOR wpp:=1 TO MAXPICKPOINT DO
	(* Verifico disponibilità Pacco *)
	IF WorkPickPointState^[wpp].State = WORKPICKPOINT_PRODOTTO_PRESENTE THEN
		(* Verifico se il codice è assegnato a qualche workarea e se la formatura è attiva *)
		FOR i:=1 TO MAXAREA DO
			IF WorkPickPointState^[wpp].Code = WorkArea^[i].Code AND WorkArea^[i].Typology = TYPOLOGY_PALLET THEN
				//CodeAssignedToWA := TRUE;
				IF WorkArea^[i].Enable = 1 AND Forming^[WorkAreaState^[i].F].Enable = 0 THEN
					TFPalletizerPackValidation := 1;//codice assegnato a workarea con formatura disabilitata
					//RETURN;
				ELSIF  WorkArea^[i].Enable = 0 AND Forming^[WorkAreaState^[i].F].Enable = 1 THEN
					TFPalletizerPackValidation := 2;//codice assegnato a workarea disabilitata
					//RETURN;
				ELSIF WorkArea^[i].Enable = 0 AND  Forming^[WorkAreaState^[i].F].Enable = 0 THEN
					TFPalletizerPackValidation := 3;//codice assegnato a workarea disabilitata e con formatura disabilitata
					//RETURN;
				ELSE
					TFPalletizerPackValidation := 0;
					//RETURN;
				END_IF
			END_IF
		END_FOR	
	END_IF
	//TFPalletizerPackValidation := 4; // Codice pacco non assegnato a nessuna workarea
END_FOR
RETURN;*)
TFPalletizerPackValidation := 0;

END_FUNCTION

// ---- POUs/TFPalletizerData/NON_USATE/TFRefreshUsedCode.TcPOU
FUNCTION TFRefreshUsedCode : BOOL
VAR_INPUT
	pcode : INT;
	UsedCode : POINTER TO ARRAY [1..MAXFORMINGCODE] OF INT;
END_VAR
VAR
	j : INT;
END_VAR

TFRefreshUsedCode := FALSE;

FOR j:=1 TO MAXFORMINGCODE-1 DO
	UsedCode^[MAXFORMINGCODE-j+1]:= UsedCode^[MAXFORMINGCODE-j];
END_FOR
UsedCode^[1] := pcode;

TFRefreshUsedCode := TRUE;

END_FUNCTION

// ---- POUs/TFPalletizerData/NON_USATE/TFWorkareaConPacchiComplete.TcPOU
FUNCTION TFWorkareaConPacchiComplete : BOOL
VAR_INPUT
	WorkArea : POINTER TO ARRAY [1..MAXAREA] OF TFMachinePalletizer_WorkArea;
	Forming : POINTER TO ARRAY [1..MAXFORMING] OF TFMachinePalletizer_Forming;
	WorkAreaState : POINTER TO ARRAY [1..MAXAREA] OF TFMachinePalletizer_WorkAreaState;
END_VAR
VAR
	wa : INT;
	n : INT;
	i : INT;
	a : INT;
END_VAR

TFWorkareaConPacchiComplete := TRUE; 

FOR wa:=1 TO MAXAREA DO
	IF WorkArea^[wa].Enable = 1 THEN
		(* Verifico se il codice è già stato assegnato *)
		IF (WorkArea^[wa].Code > 0 AND WorkArea^[wa].Typology = TYPOLOGY_PALLET) AND 
		(WorkAreaState^[wa].State < WORKAREA_STATE_OCCUPIED_WORKED AND WorkAreaState^[wa].State > WORKAREA_STATE_FREE_DISABLED) AND 
		(Forming^[WorkAreaState^[wa].F].PackXP[WorkAreaState^[wa].P].Grip <> -1 AND 
		Forming^[WorkAreaState^[wa].F].PackXN[WorkAreaState^[wa].P].Grip <> -1) THEN
			TFWorkareaConPacchiComplete := FALSE; 
			RETURN;
		END_IF
	END_IF
END_FOR

END_FUNCTION

// ---- POUs/TFPalletizerData/TFCheckPalletPresence.TcPOU
FUNCTION TFCheckPalletPresence : INT
VAR_INPUT
	WorkArea : POINTER TO ARRAY [1..MAXAREA] OF TFMachinePalletizer_WorkArea;
	WorkAreaState : POINTER TO ARRAY [1..MAXAREA] OF TFMachinePalletizer_WorkAreaState;
	PX_WorkArea : ARRAY [1..MAXAREA] OF BOOL;
END_VAR
VAR
	NStack : INT;
	i : UINT;
END_VAR

TFCheckPalletPresence := 0;
NStack := 0;

FOR i:=1 TO MAXAREAPRESENT DO
	IF WorkArea^[i].Enable = 1 AND WorkArea^[i].Typology = TYPOLOGY_STACK AND (WorkAreaState^[i].State <> WORKAREA_STATE_OCCUPIED_LGVREQ AND WorkAreaState^[i].State <> WORKAREA_STATE_OCCUPIED_LGVREQ_DISABLED) AND PX_WorkArea[i] THEN
		RETURN;
	END_IF
END_FOR
TFCheckPalletPresence := 1;

END_FUNCTION

// ---- POUs/TFPalletizerData/TFCheckLayerPresence.TcPOU
FUNCTION TFCheckLayerPresence : INT
VAR_INPUT
	WorkArea : POINTER TO ARRAY [1..MAXAREA] OF TFMachinePalletizer_WorkArea;
	WorkAreaState : POINTER TO ARRAY [1..MAXAREA] OF TFMachinePalletizer_WorkAreaState;
	PX_WorkArea : ARRAY [1..MAXAREA] OF BOOL;
END_VAR
VAR
	NStack : INT;
	i : UINT;
END_VAR

TFCheckLayerPresence := 0;
NStack := 0;

FOR i:=1 TO MAXAREAPRESENT DO
	IF WorkArea^[i].Enable = 1 AND WorkArea^[i].Typology = TYPOLOGY_LAYER AND (*WorkAreaState^[i].State = WORKAREA_STATE_OCCUPIED_WORKING*)  PX_WorkArea[i] THEN
		RETURN;
	END_IF
END_FOR
TFCheckLayerPresence := 1;

END_FUNCTION

// ---- POUs/TFPalletizerData_Lastre/Formatura/Calcolo_Formatura_Completa_24_10_2025.TcPOU
FUNCTION_BLOCK Calcolo_Formatura_Completa_24_10_2025
VAR_INPUT
	
	Supporto : TFMachinePalletizer_Pallet;
	
	//Materiale : ARRAY [0..MAXTYPE_SLABLAYER] OF Type_SlabLayer;	// Tipo di materiale, Lastra, Falda e dimensioni
	Materiale 			: ARRAY [0..MAXTYPE_SLABLAYER] OF TFMachinePalletizer_PlaceElement;	// Tipo di materiale, Lastra, Falda e dimensioni
	TipoElementoDep 	: ARRAY [1..MAXFORMINGSLAB] OF e_Tipo_Elemento_Da_Lavorare;	// Tipologia del n-esimo elemento di Materiale da depositare (Lstra-falda-terminatore)
	DimensionesPiezasLadoALadoB	: ARRAY  [1..MAXELEMENTLIST] OF ES_dimensionPiezaLadoA_ladoB;
	TipoRisultato 		: UINT := 3;// Punto utilizzato per coordinate finali di deposito lastra/falda, 1 interno, 2 centro, 3 esterno(default)
	TipoOrdinamento 	: UINT := 1;//Tipologia di ordinamento in deposito 1= alternato (lastra DX-Lastra SX), 2 = consecutivo(prima un lato, poi l'altro lato), 3 = solo lato 0°, 4 = solo lato 180°
	NumeroElementiDaDepositare : UINT;
	
	
	PulisciMemoria 				: BOOL;
	CalcolaFormatura 			: BOOL;
	In_PulisciMemoriaDone			:    BOOL;
	HabiCalTodasCordenadas: BOOL;
END_VAR

VAR_OUTPUT
	(* Variabili di uscita della posizione finale del punto di deposito della lastra/falda *)
	XFinale : ARRAY [1..MAXFORMINGSLAB] OF LREAL;		// Coordinata X punto finale n-esima lastra/falda depositata
	YFinale : ARRAY [1..MAXFORMINGSLAB] OF LREAL;		// Coordinata Y punto finale n-esima lastra/falda depositata
	ZFinale : ARRAY [1..MAXFORMINGSLAB] OF LREAL;		// Coordinata Z punto finale n-esima lastra/falda depositata
	JFinale : ARRAY [1..MAXFORMINGSLAB] OF LREAL;		// Coordinata J punto finale n-esima lastra/falda depositata
	
	XFinaleLado_0Grados : ARRAY [1..MAXFORMINGSLAB] OF LREAL;		// Coordinata X punto finale n-esima lastra/falda depositata
	YFinaleLado_0Grados : ARRAY [1..MAXFORMINGSLAB] OF LREAL;		// Coordinata Y punto finale n-esima lastra/falda depositata
	ZFinaleLado_0Grados : ARRAY [1..MAXFORMINGSLAB] OF LREAL;		// Coordinata Z punto finale n-esima lastra/falda depositata
	JFinaleLado_0Grados : ARRAY [1..MAXFORMINGSLAB] OF LREAL;		// Coordinata J punto finale n-esima lastra/falda depositata
	
	XFinaleLado_180Grados : ARRAY [1..MAXFORMINGSLAB] OF LREAL;		// Coordinata X punto finale n-esima lastra/falda depositata
	YFinaleLado_180Grados : ARRAY [1..MAXFORMINGSLAB] OF LREAL;		// Coordinata Y punto finale n-esima lastra/falda depositata
	ZFinaleLado_180Grados : ARRAY [1..MAXFORMINGSLAB] OF LREAL;		// Coordinata Z punto finale n-esima lastra/falda depositata
	JFinaleLado_180Grados : ARRAY [1..MAXFORMINGSLAB] OF LREAL;		// Coordinata J punto finale n-esima lastra/falda depositata
	
	CoorFinaleLado_Pri0_Des180 : ARRAY [1..MAXFORMINGSLAB] OF Es_CoordenadasCaballeteLadoA_ladoB ;		// Coordinata X punto finale n-esima lastra/falda depositata
	
	
	CoordenadasCaballete :  ARRAY [1..MAXFORMINGSLAB] OF Es_CoordenadasCaballeteLadoA_ladoB ;
	
	FormingSlab 			: TFMachinePalletizer_FormingForSlab;
	PulisciMemoriaDone		: BOOL;
	CalcolaFormaturaDone 	: BOOL;
	Errore 					: UINT;
END_VAR

VAR_IN_OUT
	
END_VAR

VAR
	TipoDeposito : e_TipologiaDeposito;				// ORIZZONTALE O INCLINATO
	OrdineDepositoSxDx : ARRAY [1..MAXFORMINGSLAB] OF e_Tipo_Elemento_Da_Lavorare;	// Ordine deposito materiale per i due lati, sx e dx (considero di avere il medesimo ordine di deposito dai due lati) (CAVALLINA-INCLINATO)
	
	Spessore_Lastra_Inclinata : ARRAY [1..MAXFORMINGSLAB/2] OF LREAL;				// Occupazione in larghezza della singola lastra (CAVALLINA-INCLINATO)
	Spessore_Lastra_Inclinata_Cumulato : ARRAY [1..MAXFORMINGSLAB/2] OF LREAL;	// Occupazione in larghezza delle nlastre lastre cumulate (CAVALLINA)
	Spessore_Lastra : ARRAY [1..MAXFORMINGSLAB] OF LREAL;							// Occupazione in altezza della singola lastra (CASSA-ORIZZONTALE)
	Spessore_Lastra_Cumulato : ARRAY [1..MAXFORMINGSLAB] OF LREAL;					// Occupazione in altezza delle nlastre lastre cumulate (CASSA-ORIZZONTALE)
	
	YCoordinataAppoggioLastra :  ARRAY [1..MAXFORMINGSLAB/2] OF LREAL;		// Coordinata Y del punto di appoggio della lastra sulla base della cavallina  (CAVALLINA-INCLINATO)
	ZCoordinataAppoggioLastra :  ARRAY [1..MAXFORMINGSLAB/2] OF LREAL;		// Coordinata Z del punto di appoggio della lastra sulla base della cavallina  (CAVALLINA-INCLINATO)
	
	B 	: LREAL;	// Base della cavallina (include i due lati)  (CAVALLINA-INCLINATO)
	B2	: LREAL;	// Base della cavallina (include i due lati)  (CAVALLINA-INCLINATO)
	CorYIz  : LREAL;
	CorYDe : LREAL;
	TipoCalculo : UINT := 0;
	
	BaseAlgulo : LREAL ;
	b1 : LREAL;	// base del triangolo rettangolo dell'angolo alfa  (CAVALLINA-INCLINATO)
	h1 : LREAL; // altezza del triangolo rettangolo dell'angolo alfa  (CAVALLINA-INCLINATO)
	Yd1 : ARRAY [1..MAXFORMINGSLAB/2] OF LREAL;	// Spostamento Centro lastra da inizio lastra in Y  (CAVALLINA-INCLINATO)
	Zd1 : ARRAY [1..MAXFORMINGSLAB/2] OF LREAL;	// Spostamento Centro lastra da inizio lastra in Z  (CAVALLINA-INCLINATO)
	Yd2 : ARRAY [1..MAXFORMINGSLAB/2] OF LREAL;	// Spostamento Esterno lastra da inizio lastra in Y  (CAVALLINA-INCLINATO)
	Zd2 : ARRAY [1..MAXFORMINGSLAB/2] OF LREAL;	// Spostamento Esterno lastra da inizio lastra in Z  (CAVALLINA-INCLINATOCAVALLINA)
	Yd3 : ARRAY [1..MAXFORMINGSLAB/2] OF LREAL;	// Spostamento Y dovuto al lato inclinato base appoggio  (CAVALLINA-INCLINATO)
	Zd3 : ARRAY [1..MAXFORMINGSLAB/2] OF LREAL;	// Spostamento Z dovuto al lato inclinato base appoggio  (CAVALLINA-INCLINATO)
	CI : ARRAY [1..MAXFORMINGSLAB/2] OF LREAL;	// Proiezione mancante della lastra dovuta al piano inclinato (CI) - Valorizzata solo se Beta >0  (CAVALLINA-INCLINATO)
	rad90 : LREAL;		// 90° in radianti
	
	(* Angoli piani appoggio lastre, laterale (alfa) e base (beta) cavallina *)
	AngoloAlfa_rad : LREAL;		// Angolo superiore laterale appoggio della lastra (in radianti)  (CAVALLINA-INCLINATO)
	AlgoloAlfa_gradi : LREAL; 	// Angolo superiore laterale appoggio della lastra (in gradi)  (CAVALLINA-INCLINATO)
	AngoloBeta_rad : LREAL;		// Angolo del piano inclinato di appoggio della lastra in radianti  (CAVALLINA-INCLINATO)
	AngoloBeta_gradi : LREAL; 	// Angolo del piano inclinato di appoggio della lastra in gradi  (CAVALLINA-INCLINATO)
	
	QuotaYinizioLastra : ARRAY [1..MAXFORMINGSLAB] OF LREAL;	// Quota Y inizio prima lastra  (CAVALLINA-INCLINATO)
	QuotaZinizioLastra : ARRAY [1..MAXFORMINGSLAB] OF LREAL;	// Quota Z inizio prima lastra  (CAVALLINA-INCLINATO)
	numeroLastre_int : UINT;									// Numero lastre per lato cavallina considerando la dimensione L_Utile1 (int)  (CAVALLINA-CASSA)
	
	(* Variabili di supporto *)
	counter1: UINT := 0;	// contatore per ciclo creazione formatura
	counter2: UINT := 0;	// contatore per ciclo creazione formatura
	varEven : UINT := 0;	// Pari o dispari per lato destro (dispari) o lato sinistro (pari) cavallina
	
	(* Variabili di uscita della posizione del punto interno, centrale ed esterno della lastra *)
	XInternoLastra : ARRAY [1..MAXFORMINGSLAB] OF LREAL;		// Coordinata X punto interno n-esima lastra depositata  (CAVALLINA-CASSA)
	YInternoLastra : ARRAY [1..MAXFORMINGSLAB] OF LREAL;		// Coordinata Y punto interno n-esima lastra depositata  (CAVALLINA-CASSA)
	ZInternoLastra : ARRAY [1..MAXFORMINGSLAB] OF LREAL;		// Coordinata Z punto interno n-esima lastra depositata  (CAVALLINA-CASSA)
	XCentroLastra  : ARRAY [1..MAXFORMINGSLAB] OF LREAL;		// Coordinata X punto centrale n-esima lastra depositata  (CAVALLINA-CASSA)
	YCentroLastra  : ARRAY [1..MAXFORMINGSLAB] OF LREAL;		// Coordinata Y punto centrale n-esima lastra depositata  (CAVALLINA-CASSA)
	ZCentroLastra  : ARRAY [1..MAXFORMINGSLAB] OF LREAL;		// Coordinata Z punto centrale n-esima lastra depositata  (CAVALLINA-CASSA)
	XEsternoLastra : ARRAY [1..MAXFORMINGSLAB] OF LREAL;		// Coordinata X punto esterno n-esima lastra depositata  (CAVALLINA-CASSA)
	YEsternoLastra : ARRAY [1..MAXFORMINGSLAB] OF LREAL;		// Coordinata Y punto esterno n-esima lastra depositata  (CAVALLINA-CASSA)
	ZEsternoLastra : ARRAY [1..MAXFORMINGSLAB] OF LREAL;		// Coordinata Z punto esterno n-esima lastra depositata  (CAVALLINA-CASSA)

	P_TextModeWrite : P_TextModeWrite;
	MemoriaInizializzata 		:    BOOL;
	NuPiezasLadoDx : INT ;
	NuPiezasLadoSx : INT ;
	CalForCavallete: UINT;
	F_ini: UINT;
	F_Fin: UINT;
	
	CntLados: UINT;
END_VAR

VAR CONSTANT
END_VAR

// Pulisco le variabili interne e le variabili di uscita del FB
IF PulisciMemoria AND NOT PulisciMemoriaDone THEN		// Pulizia delle variabili locali e di uscita
	PulisciMemoriaDone := TRUE;
	memset(ADR(XFinale), 0 , SIZEOF(XFinale));memset(ADR(YFinale), 0 , SIZEOF(YFinale));memset(ADR(ZFinale), 0 , SIZEOF(ZFinale));memset(ADR(JFinale), 0 , SIZEOF(JFinale));
	//###########################################
	memset(ADR(XFinaleLado_0Grados), 0 , SIZEOF(XFinaleLado_0Grados));memset(ADR(YFinaleLado_0Grados), 0 , SIZEOF(YFinaleLado_0Grados));memset(ADR(ZFinaleLado_0Grados), 0 , SIZEOF(ZFinaleLado_0Grados));memset(ADR(JFinaleLado_0Grados), 0 , SIZEOF(JFinaleLado_0Grados));
	memset(ADR(XFinaleLado_180Grados), 0 , SIZEOF(XFinaleLado_180Grados));memset(ADR(YFinaleLado_180Grados), 0 , SIZEOF(YFinaleLado_180Grados));memset(ADR(ZFinaleLado_180Grados), 0 , SIZEOF(ZFinaleLado_180Grados));memset(ADR(JFinaleLado_180Grados), 0 , SIZEOF(JFinaleLado_180Grados));
	memset(ADR(CoorFinaleLado_Pri0_Des180), 0 , SIZEOF(CoorFinaleLado_Pri0_Des180));
	//###########################################################################################
	memset(ADR(FormingSlab), 0 , SIZEOF(FormingSlab));
	memset(ADR(Errore), 0 , SIZEOF(Errore));
	memset(ADR(OrdineDepositoSxDx), 0 , SIZEOF(OrdineDepositoSxDx));
	memset(ADR(Spessore_Lastra_Inclinata), 0 , SIZEOF(Spessore_Lastra_Inclinata));memset(ADR(Spessore_Lastra_Inclinata_Cumulato), 0 , SIZEOF(Spessore_Lastra_Inclinata_Cumulato));
	memset(ADR(Spessore_Lastra), 0 , SIZEOF(Spessore_Lastra));memset(ADR(Spessore_Lastra_Cumulato), 0 , SIZEOF(Spessore_Lastra_Cumulato));
	memset(ADR(YCoordinataAppoggioLastra), 0 , SIZEOF(YCoordinataAppoggioLastra));memset(ADR(ZCoordinataAppoggioLastra), 0 , SIZEOF(ZCoordinataAppoggioLastra));
	memset(ADR(B), 0 , SIZEOF(B));memset(ADR(b1), 0 , SIZEOF(b1));memset(ADR(h1), 0 , SIZEOF(h1));
	memset(ADR(Yd1), 0 , SIZEOF(Yd1));memset(ADR(Zd1), 0 , SIZEOF(Zd1));
	memset(ADR(Yd2), 0 , SIZEOF(Yd2));memset(ADR(Zd2), 0 , SIZEOF(Zd2));
	memset(ADR(Yd3), 0 , SIZEOF(Yd3));memset(ADR(Zd3), 0 , SIZEOF(Zd3));
	memset(ADR(CI), 0 , SIZEOF(CI));
	memset(ADR(AngoloAlfa_rad), 0 , SIZEOF(AngoloAlfa_rad));memset(ADR(AngoloBeta_rad), 0 , SIZEOF(AngoloBeta_rad));
	memset(ADR(QuotaYinizioLastra), 0 , SIZEOF(QuotaYinizioLastra));memset(ADR(QuotaZinizioLastra), 0 , SIZEOF(QuotaZinizioLastra));
	memset(ADR(numeroLastre_int), 0 , SIZEOF(numeroLastre_int));
	memset(ADR(XInternoLastra), 0 , SIZEOF(XInternoLastra));memset(ADR(YInternoLastra), 0 , SIZEOF(YInternoLastra));memset(ADR(ZInternoLastra), 0 , SIZEOF(ZInternoLastra));
	memset(ADR(XCentroLastra), 0 , SIZEOF(XCentroLastra));memset(ADR(YCentroLastra), 0 , SIZEOF(YCentroLastra));memset(ADR(ZCentroLastra), 0 , SIZEOF(ZCentroLastra));
	memset(ADR(XEsternoLastra), 0 , SIZEOF(XEsternoLastra));memset(ADR(YEsternoLastra), 0 , SIZEOF(YEsternoLastra));memset(ADR(ZEsternoLastra), 0 , SIZEOF(ZEsternoLastra));
	memset(ADR(Supporto), 0 , SIZEOF(Supporto));
	memset(ADR(Materiale), 0 , SIZEOF(Materiale));
	memset(ADR(TipoElementoDep), 99 , SIZEOF(TipoElementoDep));
	Errore := 0;
	HabiCalTodasCordenadas := FALSE ;
	MemoriaInizializzata := TRUE;
ELSIF NOT PulisciMemoria AND PulisciMemoriaDone THEN
	PulisciMemoriaDone := FALSE;
END_IF

// Calcolo la Formatura, tipo Cassa o Cavallina e salvo su file i risultati ottenuti
IF CalcolaFormatura AND NOT CalcolaFormaturaDone AND MemoriaInizializzata THEN
	// Pulisco le variabili interne e le variabili di uscita del FB
	memset(ADR(XFinale), 0 , SIZEOF(XFinale));memset(ADR(YFinale), 0 , SIZEOF(YFinale));memset(ADR(ZFinale), 0 , SIZEOF(ZFinale));memset(ADR(JFinale), 0 , SIZEOF(JFinale));
	memset(ADR(FormingSlab), 0 , SIZEOF(FormingSlab));
	memset(ADR(Errore), 0 , SIZEOF(Errore));
	memset(ADR(OrdineDepositoSxDx), 0 , SIZEOF(OrdineDepositoSxDx));
	memset(ADR(Spessore_Lastra_Inclinata), 0 , SIZEOF(Spessore_Lastra_Inclinata));memset(ADR(Spessore_Lastra_Inclinata_Cumulato), 0 , SIZEOF(Spessore_Lastra_Inclinata_Cumulato));
	memset(ADR(Spessore_Lastra), 0 , SIZEOF(Spessore_Lastra));memset(ADR(Spessore_Lastra_Cumulato), 0 , SIZEOF(Spessore_Lastra_Cumulato));
	memset(ADR(YCoordinataAppoggioLastra), 0 , SIZEOF(YCoordinataAppoggioLastra));memset(ADR(ZCoordinataAppoggioLastra), 0 , SIZEOF(ZCoordinataAppoggioLastra));
	memset(ADR(B), 0 , SIZEOF(B));memset(ADR(b1), 0 , SIZEOF(b1));memset(ADR(h1), 0 , SIZEOF(h1));
	memset(ADR(Yd1), 0 , SIZEOF(Yd1));memset(ADR(Zd1), 0 , SIZEOF(Zd1));
	memset(ADR(Yd2), 0 , SIZEOF(Yd2));memset(ADR(Zd2), 0 , SIZEOF(Zd2));
	memset(ADR(Yd3), 0 , SIZEOF(Yd3));memset(ADR(Zd3), 0 , SIZEOF(Zd3));
	memset(ADR(CI), 0 , SIZEOF(CI));
	memset(ADR(AngoloAlfa_rad), 0 , SIZEOF(AngoloAlfa_rad));memset(ADR(AngoloBeta_rad), 0 , SIZEOF(AngoloBeta_rad));
	memset(ADR(QuotaYinizioLastra), 0 , SIZEOF(QuotaYinizioLastra));memset(ADR(QuotaZinizioLastra), 0 , SIZEOF(QuotaZinizioLastra));
	memset(ADR(numeroLastre_int), 0 , SIZEOF(numeroLastre_int));
	memset(ADR(XInternoLastra), 0 , SIZEOF(XInternoLastra));memset(ADR(YInternoLastra), 0 , SIZEOF(YInternoLastra));memset(ADR(ZInternoLastra), 0 , SIZEOF(ZInternoLastra));
	memset(ADR(XCentroLastra), 0 , SIZEOF(XCentroLastra));memset(ADR(YCentroLastra), 0 , SIZEOF(YCentroLastra));memset(ADR(ZCentroLastra), 0 , SIZEOF(ZCentroLastra));
	memset(ADR(XEsternoLastra), 0 , SIZEOF(XEsternoLastra));memset(ADR(YEsternoLastra), 0 , SIZEOF(YEsternoLastra));memset(ADR(ZEsternoLastra), 0 , SIZEOF(ZEsternoLastra));

	// Definizione del tipo di deposito a seconda del tipo di supporto utilizzato
	CASE Supporto.Tipologia OF
		PALLET_STANDARD : TipoDeposito := ORIZZONTALE;
		CASSA_STANDARD 	: TipoDeposito := ORIZZONTALE;
		CAVALLETTO 		: TipoDeposito := INCLINATO ; TipoRisultato := TipoLLenarCavellete ;
		BUNDLE 			: TipoDeposito := INCLINATO ; TipoRisultato := TipoLLenarCavellete;//INCLINATO_LATOSINGOLO;
	END_CASE
	
	CASE TipoDeposito OF
		ORIZZONTALE:				// Tipo deposito Orizzontale (Cassa o Pallet)
			(* CASO DELLA CASSA/PALLET CON DEPOSITO ORIZZONTALE *)
			
			(* Creo un ordine di deposito generico, per effettuare i test del singolo lato della cavallina, per debug  *)
			numeroLastre_int := 0;
			FOR counter1:=1 TO MAXFORMINGSLAB BY 1 DO
				IF (TipoElementoDep[counter1] <> e_Tipo_Elemento_Da_Lavorare.NOT_DEFINED AND TipoElementoDep[counter1] <> TERMINATORE) THEN
					numeroLastre_int := numeroLastre_int+1;
				END_IF;
			END_FOR
			
			(* Controlli dati coerenti *)
			IF (Supporto.HMAX <= 0 ) 	OR (Supporto.YDim <= 0 ) THEN
				Errore := ErrValori;
			END_IF
			
			IF (Supporto.ZDim <= 0) THEN
				Errore := ErrHBaseInternaNulla;
				RETURN;
			END_IF
			
			IF (Supporto.XDim <= 0) THEN
				Errore := ErroreLBaseNulla;
				RETURN;
			END_IF
			
			FOR counter1 :=1 TO numeroLastre_int DO
				IF (Supporto.YDim+30 <= Materiale[TipoElementoDep[counter1]].YDim) OR (Supporto.XDim+30 <= Materiale[TipoElementoDep[counter1]].XDim) THEN
					Errore := ErrDimensioneCassa;
				RETURN;
				END_IF
			END_FOR
			
			memset(ADR(Spessore_Lastra), 0 , SIZEOF(Spessore_Lastra));
			FOR counter2 := 1 TO MAXFORMINGSLAB BY 1 DO
				Spessore_Lastra[counter2] := Materiale[TipoElementoDep[counter2]].ZDim;
			END_FOR
			
			// Calcola lo spessore complessivo fino al passo n delle lastre/falde depositate sul singolo lato della cavallina 
			memset(ADR(Spessore_Lastra_Cumulato), 0 , SIZEOF(Spessore_Lastra_Cumulato));
			IF (Spessore_Lastra_Cumulato[1] = 0) THEN
				FOR counter2:=1 TO MAXFORMINGSLAB BY 1 DO
					FOR counter1 := 1 TO counter2 BY 1 DO
						Spessore_Lastra_Cumulato[counter2] := Spessore_Lastra_Cumulato[counter2] + Spessore_Lastra[counter1];
					END_FOR
				END_FOR
			END_IF
			
			// Numero di possibili lastre sulla cassa (minore dell'altezza massima)
			FOR counter1:=1 TO MAXFORMINGSLAB BY 1 DO
				IF (TipoElementoDep[counter1] <> e_Tipo_Elemento_Da_Lavorare.NOT_DEFINED AND TipoElementoDep[counter1] <> TERMINATORE) AND ((Spessore_Lastra_Cumulato[counter1] >0) AND 
					(Spessore_Lastra_Cumulato[counter1]+Supporto.ZDim < Supporto.HMAX)) THEN
						numeroLastre_int := counter1;
				END_IF
				IF (Spessore_Lastra_Cumulato[counter1]+Supporto.ZDim >= Supporto.HMAX) AND Supporto.Tipologia <> PALLET_STANDARD AND counter1 <= numeroLastre_int THEN
					Errore := ErrNumeroPezzi;
				END_IF
			END_FOR
			
			// Calcolo il punto Z interno, centrale ed esterno per ogni lastra posizionata sulla cassa
			FOR counter1:=1 TO numeroLastre_int BY 1 DO
				ZInternoLastra[counter1] := Supporto.ZDim + Spessore_Lastra_Cumulato[counter1-1];
				ZCentroLastra[counter1] := Supporto.ZDim + (Spessore_Lastra_Cumulato[counter1-1] + Spessore_Lastra_Cumulato[counter1]) / 2;
				ZEsternoLastra[counter1] := Supporto.ZDim + Spessore_Lastra_Cumulato[counter1];
			END_FOR
			
			(* Pulisco le uscite e setto a TERMINATORE tutti gli elementi di FormingSlab *)
			memset(ADR(XFinale),0,SIZEOF(XFinale));memset(ADR(YFinale),0,SIZEOF(YFinale));memset(ADR(ZFinale),0,SIZEOF(ZFinale));memset(ADR(JFinale),0,SIZEOF(JFinale));
			memset(ADR(FormingSlab),0,SIZEOF(FormingSlab));
			FOR counter1 := 1 TO MAXFORMINGSLAB DO
				FormingSlab.PElement[counter1].Typology := TERMINATORE;
			END_FOR
			
			(* Calcolo delle coordinate X,Y,Z del punto finale sulla base del TipoRisultato *)
			FOR counter2:=1 TO numeroLastre_int BY 1 DO
				XInternoLastra[counter2] := 0; YInternoLastra[counter2] := 0;
				XCentroLastra[counter2] := 0;  YCentroLastra[counter2] := 0;
				XEsternoLastra[counter2] := 0; YEsternoLastra[counter2] := 0;
				
				CASE TipoRisultato OF
					1:	XFinale[counter2] := XInternoLastra[counter2] + Supporto.OFSDE_X90;
						YFinale[counter2] := YInternoLastra[counter2] + Supporto.OFSDE_Y90;
						ZFinale[counter2] := ZInternoLastra[counter2] + Supporto.OFSDE_Z90;
						JFinale[counter2] := 90 + Supporto.OFSDE_J90;
					2:	XFinale[counter2] := XCentroLastra[counter2] + Supporto.OFSDE_X90;
						YFinale[counter2] := YCentroLastra[counter2] + Supporto.OFSDE_Y90;
						ZFinale[counter2] := ZCentroLastra[counter2] + Supporto.OFSDE_Z90;
						JFinale[counter2] := 90  + Supporto.OFSDE_J90;
					3:	XFinale[counter2] := XEsternoLastra[counter2] + Supporto.OFSDE_X90;
						YFinale[counter2] := YEsternoLastra[counter2] + Supporto.OFSDE_Y90;
						ZFinale[counter2] := ZEsternoLastra[counter2] + Supporto.OFSDE_Z90;
						JFinale[counter2] := 90 + Supporto.OFSDE_J90;	
				END_CASE
				
			END_FOR;
			FOR counter1:=1 TO numeroLastre_int BY 1 DO
				FormingSlab.Enable := 1;										// Abilitato
				//FormingSlab.Code[1] := 1;
				//FormingSlab.PElement[counter1].Typology := Materiale[OrdineDeposito[counter1]].Typology;

				//Indico la tipologia di elemnto che vado a depositare in base all'ordine passato dall'esterno
				CASE TipoElementoDep[counter1] OF
					LASTRA:
						FormingSlab.PElement[counter1].Typology := LASTRA;

					FALDA:
						FormingSlab.PElement[counter1].Typology := FALDA;

					TERMINATORE:
						FormingSlab.PElement[counter1].Typology := TERMINATORE;
				
				ELSE
					FormingSlab.PElement[counter1].Typology := e_Tipo_Elemento_Da_Lavorare.NOT_DEFINED;

				END_CASE
				
				FormingSlab.PElement[counter1].XDim := Materiale[TipoElementoDep[counter1]].XDim;		// Dimensione X Lastra		
				FormingSlab.PElement[counter1].YDim := Materiale[TipoElementoDep[counter1]].YDim;		// Dimensione Y Lastra
				FormingSlab.PElement[counter1].ZDim := Materiale[TipoElementoDep[counter1]].ZDim;		// Dimensione Z Lastra
				FormingSlab.PElement[counter1].X := XFinale[counter1];
				FormingSlab.PElement[counter1].Y := YFinale[counter1];
				FormingSlab.PElement[counter1].Z := ZFinale[counter1];
				FormingSlab.PElement[counter1].J := JFinale[counter1];
			END_FOR
		
			
		
		INCLINATO:					// Tipo deposito inclinato ( Cavallina)
			(* CASO DELLA CAVALLINA CON DEPOSITO INCLINATO DAI DUE LATI*)
			
			numeroLastre_int := 0;
			FOR counter1:=1 TO MAXFORMINGSLAB/2 BY 1 DO
				IF (TipoElementoDep[counter1] <> e_Tipo_Elemento_Da_Lavorare.NOT_DEFINED AND TipoElementoDep[counter1] <> TERMINATORE) THEN
					numeroLastre_int := numeroLastre_int+1;
				END_IF;
			END_FOR
	
			(* Replico l'ordine di deposito del singolo lato su entrambi i lati, sx e dx della cavallina *)
			FOR counter1:=1 TO MAXFORMINGSLAB BY 1 DO
				varEven := counter1 MOD 2;
				CASE varEven OF
					0:	
						OrdineDepositoSxDx[counter1] := TipoElementoDep[counter1];//OrdineDeposito[counter1/2];
					1:	
						OrdineDepositoSxDx[counter1] := TipoElementoDep[counter1];//OrdineDeposito[(counter1+varEven)/2];
				END_CASE;
			END_FOR;
			
			(* Controlli dati coerenti *)
			FOR counter1:=1 TO MAXFORMINGSLAB DO
				IF(Materiale[TipoElementoDep[counter1]].XDim <0) OR (Materiale[TipoElementoDep[counter1]].YDim <0) OR 
					(Materiale[TipoElementoDep[counter1]].ZDim <0)  OR (Materiale[TipoElementoDep[counter1]].Typology <0) THEN
						Errore := Errvalori;
						RETURN;
				END_IF
			END_FOR
					
			IF Supporto.ZDim <= 0 THEN//OR (Supporto.ZDim_Int2 <=0) THEN
				Errore := ErrHBaseInternaNulla;
				RETURN;
			END_IF
			
			IF Supporto.ZDim_Ext1 <= 0 AND Supporto.TipoPianoAppoggio = 1 THEN//OR (Supporto.ZDim_Ext2 <=0) THEN
				Errore := ErrHBaseEsternaNulla;
				RETURN;
			END_IF
			
			IF Supporto.ZDim > Supporto.ZDim_Ext1 AND Supporto.TipoPianoAppoggio = 1 THEN//OR (Supporto.ZDim_Int2 > Supporto.ZDim_Ext2) THEN
				Errore := ErrBaseInclinata;
				RETURN;
			END_IF
			
			IF (Supporto.HMAX <= 0) THEN		// altezza cavallina
				Errore := ErrHTotaleNulla;
				RETURN;
			END_IF
			
			IF (Supporto.YDim <= 0) THEN		// larghezza Y cavallina
				Errore := ErroreLBaseNulla;
				RETURN;
			END_IF
			
